Yaskawa INFORM job: DEMO_ROOF_SIDE_0625_3PAINT_51.JBI

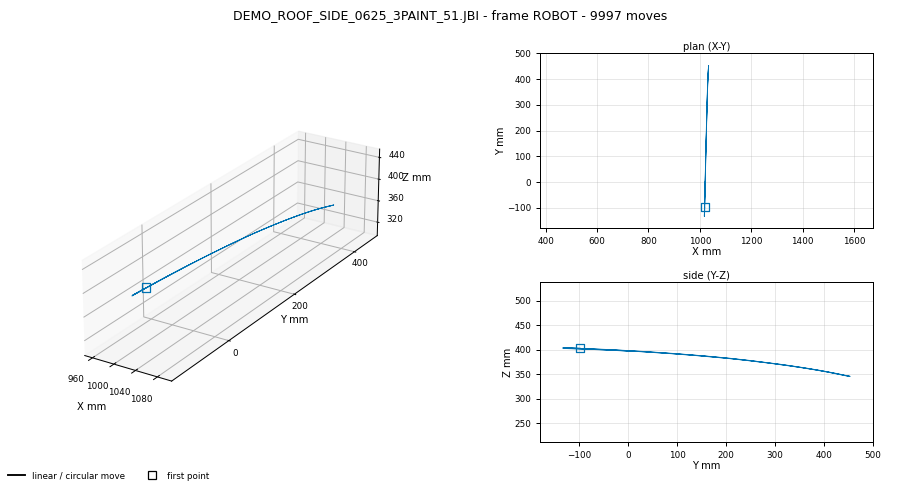
[picture p0: tool path of DEMO_ROOF_SIDE_0625_3PAINT_51.JBI in frame ROBOT, 9997 of 9997 moves have a stored position in this frame; points joined in program order, loops and branches not executed]
/JOB
//NAME DEMO_ROOF_SIDE_0625_3PAINT51
//POS
///NPOS 9997,0,0,0,0,0
///TOOL 0
///USER 0
///POSTYPE ROBOT
///RECTAN
///RCONF 1,0,0,0,0,0,0,0,0,0,0,0,0,0,0,0,0,0,0,0,0,0,0,0
C00000=1018.937,-97.840,403.399,165.576,52.819,159.418
C00001=1018.932,-98.090,403.408,165.573,52.823,159.418
C00002=1018.926,-98.340,403.416,165.570,52.828,159.419
C00003=1018.920,-98.590,403.426,165.567,52.833,159.419
C00004=1018.915,-98.839,403.434,165.564,52.838,159.419
C00005=1018.910,-99.089,403.443,165.561,52.842,159.419
C00006=1018.905,-99.339,403.452,165.558,52.848,159.420
C00007=1018.900,-99.589,403.460,165.555,52.852,159.420
C00008=1018.894,-99.839,403.469,165.552,52.857,159.420
C00009=1018.888,-100.088,403.478,165.549,52.862,159.420
C00010=1018.883,-100.338,403.487,165.546,52.867,159.420
C00011=1018.878,-100.588,403.495,165.542,52.871,159.421
C00012=1018.873,-100.837,403.504,165.540,52.876,159.421
C00013=1018.867,-101.087,403.512,165.537,52.881,159.421
C00014=1018.861,-101.371,403.523,165.534,52.887,159.421
C00015=1018.856,-101.655,403.533,165.531,52.892,159.422
C00016=1018.850,-101.939,403.543,165.526,52.897,159.422
C00017=1018.844,-102.223,403.552,165.523,52.902,159.422
C00018=1018.838,-102.472,403.561,165.520,52.908,159.422
C00019=1018.833,-102.722,403.570,165.517,52.912,159.423
C00020=1018.827,-102.972,403.579,165.514,52.917,159.423
C00021=1018.822,-103.222,403.587,165.510,52.921,159.423
C00022=1018.817,-103.472,403.596,165.508,52.927,159.423
C00023=1018.811,-103.721,403.604,165.505,52.931,159.423
C00024=1018.806,-103.971,403.613,165.501,52.936,159.424
C00025=1018.801,-104.221,403.621,165.499,52.940,159.424
C00026=1018.796,-104.471,403.630,165.496,52.946,159.424
C00027=1018.791,-104.720,403.639,165.492,52.950,159.424
C00028=1018.786,-104.970,403.647,165.490,52.955,159.425
C00029=1018.781,-105.220,403.656,165.486,52.959,159.425
C00030=1018.775,-105.470,403.664,165.483,52.965,159.425
C00031=1018.770,-105.720,403.673,165.481,52.969,159.425
C00032=1018.764,-105.970,403.681,165.477,52.974,159.425
C00033=1018.759,-106.219,403.690,165.475,52.978,159.426
C00034=1018.754,-106.469,403.698,165.472,52.984,159.426
C00035=1018.748,-106.719,403.707,165.468,52.988,159.426
C00036=1018.743,-106.969,403.715,165.466,52.993,159.426
C00037=1018.738,-107.219,403.723,165.462,52.997,159.426
C00038=1018.733,-107.469,403.732,165.459,53.003,159.427
C00039=1018.728,-107.718,403.740,165.457,53.007,159.427
C00040=1018.722,-107.968,403.749,165.453,53.012,159.427
///RCONF 1,0,0,0,1,0,0,0,0,0,0,0,0,0,0,0,0,0,0,0,0,0,0,0
C00041=1018.717,-108.218,403.757,165.450,53.017,159.427
C00042=1018.712,-108.468,403.766,165.448,53.022,159.428
C00043=1018.707,-108.718,403.773,165.444,53.026,159.428
C00044=1018.702,-108.968,403.782,165.441,53.032,159.428
C00045=1018.696,-109.217,403.790,165.439,53.036,159.428
C00046=1018.691,-109.467,403.799,165.435,53.041,159.429
C00047=1018.686,-109.717,403.807,165.432,53.045,159.429
C00048=1018.680,-109.967,403.814,165.429,53.051,159.429
C00049=1018.675,-110.216,403.823,165.426,53.055,159.429
C00050=1018.670,-110.466,403.831,165.423,53.060,159.429
C00051=1018.664,-110.716,403.840,165.420,53.065,159.430
C00052=1018.660,-110.966,403.847,165.417,53.070,159.430
C00053=1018.655,-111.215,403.856,165.414,53.074,159.430
C00054=1018.650,-111.465,403.864,165.411,53.080,159.430
C00055=1018.645,-111.715,403.872,165.408,53.084,159.431
C00056=1018.639,-111.965,403.880,165.405,53.089,159.431
C00057=1018.634,-112.215,403.889,165.401,53.094,159.431
C00058=1018.628,-112.464,403.897,165.399,53.099,159.431
C00059=1018.623,-112.714,403.905,165.396,53.103,159.431
C00060=1018.618,-112.964,403.913,165.392,53.108,159.432
C00061=1018.613,-113.214,403.922,165.390,53.112,159.432
C00062=1018.608,-113.464,403.929,165.387,53.118,159.432
C00063=1018.603,-113.713,403.938,165.384,53.122,159.432
C00064=1018.598,-113.964,403.945,165.381,53.127,159.432
C00065=1018.593,-114.213,403.954,165.377,53.132,159.433
C00066=1018.587,-114.463,403.962,165.375,53.137,159.433
C00067=1018.582,-114.713,403.969,165.372,53.141,159.433
C00068=1018.576,-114.963,403.978,165.368,53.146,159.433
C00069=1018.571,-115.213,403.986,165.366,53.151,159.434
C00070=1018.567,-115.462,403.994,165.363,53.156,159.434
C00071=1018.561,-115.712,404.001,165.359,53.161,159.434
C00072=1018.556,-115.962,404.009,165.357,53.166,159.434
C00073=1018.551,-116.212,404.018,165.354,53.170,159.435
C00074=1018.546,-116.462,404.026,165.350,53.175,159.435
C00075=1018.540,-116.711,404.033,165.347,53.180,159.435
C00076=1018.535,-116.961,404.041,165.345,53.185,159.435
C00077=1018.530,-117.211,404.049,165.341,53.190,159.435
C00078=1018.524,-117.495,404.059,165.338,53.195,159.436
C00079=1018.518,-117.779,404.067,165.335,53.201,159.436
C00080=1018.513,-118.062,404.076,165.331,53.206,159.436
C00081=1018.507,-118.346,404.085,165.328,53.211,159.436
C00082=1018.502,-118.596,404.092,165.325,53.216,159.437
C00083=1018.496,-118.846,404.101,165.322,53.221,159.437
C00084=1018.491,-119.095,404.108,165.319,53.226,159.437
C00085=1018.486,-119.345,404.116,165.316,53.231,159.437
C00086=1018.481,-119.595,404.124,165.313,53.235,159.437
C00087=1018.475,-119.845,404.131,165.310,53.240,159.438
C00088=1018.471,-120.094,404.139,165.307,53.246,159.438
C00089=1018.466,-120.345,404.147,165.304,53.250,159.438
C00090=1018.460,-120.594,404.155,165.301,53.255,159.438
C00091=1018.455,-120.844,404.163,165.297,53.259,159.438
C00092=1018.450,-121.094,404.170,165.295,53.264,159.439
C00093=1018.445,-121.344,404.179,165.292,53.269,159.439
C00094=1018.439,-121.594,404.186,165.288,53.274,159.439
C00095=1018.435,-121.843,404.193,165.286,53.278,159.439
C00096=1018.430,-122.094,404.201,165.283,53.284,159.440
C00097=1018.424,-122.343,404.209,165.279,53.288,159.440
C00098=1018.420,-122.593,404.216,165.277,53.293,159.440
C00099=1018.415,-122.843,404.224,165.274,53.298,159.440
C00100=1018.409,-123.093,404.232,165.270,53.303,159.440
C00101=1018.404,-123.342,404.239,165.268,53.307,159.441
C00102=1018.399,-123.593,404.247,165.264,53.312,159.441
C00103=1018.394,-123.843,404.254,165.261,53.318,159.441
C00104=1018.389,-124.092,404.262,165.259,53.322,159.441
C00105=1018.383,-124.342,404.269,165.255,53.327,159.441
C00106=1018.378,-124.592,404.277,165.253,53.331,159.442
C00107=1018.374,-124.842,404.285,165.250,53.337,159.442
C00108=1018.368,-125.092,404.292,165.246,53.341,159.442
C00109=1018.363,-125.342,404.300,165.244,53.346,159.442
C00110=1018.358,-125.591,404.307,165.241,53.351,159.443
C00111=1018.353,-125.841,404.315,165.238,53.356,159.443
C00112=1018.348,-126.090,404.322,165.235,53.360,159.443
C00113=1018.343,-126.341,404.329,165.232,53.366,159.443
C00114=1018.337,-126.591,404.337,165.229,53.370,159.443
C00115=1018.333,-126.840,404.344,165.225,53.375,159.443
C00116=1018.327,-127.090,404.351,165.223,53.380,159.444
C00117=1018.323,-127.340,404.359,165.220,53.385,159.444
C00118=1018.317,-127.590,404.366,165.217,53.389,159.444
C00119=1018.313,-127.839,404.374,165.214,53.394,159.444
C00120=1018.307,-128.089,404.381,165.211,53.400,159.445
C00121=1018.302,-128.339,404.389,165.208,53.403,159.445
C00122=1018.299,-128.588,404.397,165.205,53.408,159.445
C00123=1018.295,-128.837,404.406,165.202,53.410,159.445
C00124=1018.291,-129.088,404.416,165.200,53.413,159.445
C00125=1018.288,-129.337,404.426,165.196,53.416,159.444
C00126=1018.285,-129.586,404.437,165.195,53.417,159.444
C00127=1018.283,-129.836,404.448,165.192,53.418,159.444
C00128=1018.282,-130.086,404.460,165.190,53.419,159.444
C00129=1018.280,-130.336,404.473,165.187,53.419,159.443
C00130=1018.279,-130.586,404.486,165.184,53.419,159.443
C00131=1018.279,-130.836,404.500,165.182,53.418,159.442
C00132=1018.278,-131.085,404.514,165.180,53.416,159.441
C00133=1018.279,-131.334,404.529,165.178,53.414,159.440
C00134=1018.280,-131.584,404.545,165.176,53.412,159.440
C00135=1018.281,-131.834,404.560,165.174,53.408,159.438
C00136=1018.283,-132.083,404.577,165.172,53.406,159.438
C00137=1018.285,-132.333,404.594,165.170,53.401,159.436
C00138=1018.288,-132.583,404.612,165.168,53.396,159.435
C00139=1018.290,-132.833,404.631,165.167,53.391,159.434
C00140=1018.294,-133.082,404.650,165.165,53.385,159.432
C00141=1018.298,-133.332,404.669,165.164,53.379,159.431
C00142=1018.032,-133.358,404.292,165.121,53.715,159.480
C00143=1018.028,-133.109,404.273,165.123,53.722,159.482
C00144=1018.026,-132.859,404.255,165.125,53.727,159.483
C00145=1018.022,-132.610,404.236,165.127,53.732,159.485
C00146=1018.020,-132.360,404.218,165.128,53.737,159.486
C00147=1018.018,-132.110,404.201,165.130,53.742,159.487
C00148=1018.017,-131.860,404.184,165.132,53.746,159.488
C00149=1018.015,-131.610,404.168,165.134,53.748,159.489
C00150=1018.014,-131.361,404.152,165.135,53.751,159.490
C00151=1018.013,-131.111,404.137,165.138,53.753,159.490
C00152=1018.014,-130.861,404.123,165.140,53.754,159.491
C00153=1018.014,-130.611,404.109,165.142,53.755,159.492
C00154=1018.015,-130.362,404.096,165.145,53.755,159.492
C00155=1018.016,-130.112,404.084,165.147,53.755,159.493
C00156=1018.018,-129.862,404.072,165.150,53.755,159.493
C00157=1018.020,-129.613,404.060,165.153,53.754,159.494
C00158=1018.023,-129.363,404.050,165.154,53.752,159.494
C00159=1018.026,-129.113,404.039,165.158,53.749,159.494
C00160=1018.029,-128.864,404.030,165.160,53.747,159.494
C00161=1018.033,-128.614,404.021,165.163,53.743,159.494
C00162=1018.037,-128.365,404.012,165.166,53.739,159.494
C00163=1018.042,-128.115,404.004,165.168,53.735,159.494
C00164=1018.046,-127.866,403.996,165.172,53.730,159.494
C00165=1018.052,-127.616,403.989,165.175,53.725,159.494
C00166=1018.057,-127.366,403.982,165.178,53.720,159.493
C00167=1018.061,-127.117,403.975,165.180,53.716,159.493
C00168=1018.067,-126.867,403.968,165.183,53.710,159.493
C00169=1018.072,-126.616,403.960,165.187,53.705,159.493
C00170=1018.077,-126.367,403.953,165.190,53.700,159.493
C00171=1018.082,-126.117,403.945,165.192,53.695,159.492
C00172=1018.087,-125.867,403.939,165.196,53.691,159.492
C00173=1018.092,-125.617,403.931,165.199,53.685,159.492
C00174=1018.098,-125.368,403.923,165.202,53.680,159.492
C00175=1018.103,-125.118,403.915,165.204,53.675,159.491
C00176=1018.108,-124.868,403.908,165.208,53.670,159.491
C00177=1018.113,-124.618,403.901,165.211,53.666,159.491
C00178=1018.118,-124.368,403.893,165.214,53.660,159.491
C00179=1018.123,-124.119,403.886,165.216,53.656,159.490
C00180=1018.128,-123.868,403.879,165.220,53.651,159.490
C00181=1018.133,-123.619,403.870,165.223,53.645,159.490
C00182=1018.138,-123.369,403.863,165.225,53.641,159.490
C00183=1018.143,-123.119,403.856,165.229,53.636,159.490
C00184=1018.148,-122.869,403.848,165.232,53.631,159.489
C00185=1018.153,-122.620,403.840,165.235,53.626,159.489
C00186=1018.158,-122.370,403.832,165.237,53.621,159.489
C00187=1018.163,-122.119,403.825,165.241,53.616,159.489
C00188=1018.168,-121.870,403.818,165.244,53.611,159.489
C00189=1018.174,-121.620,403.809,165.246,53.606,159.488
C00190=1018.179,-121.370,403.802,165.249,53.602,159.488
C00191=1018.184,-121.121,403.795,165.253,53.597,159.488
C00192=1018.189,-120.870,403.787,165.256,53.591,159.488
C00193=1018.194,-120.621,403.779,165.258,53.587,159.487
C00194=1018.199,-120.371,403.772,165.261,53.581,159.487
C00195=1018.207,-119.987,403.759,165.266,53.574,159.487
C00196=1018.215,-119.603,403.748,165.271,53.566,159.487
C00197=1018.223,-119.219,403.735,165.275,53.559,159.486
C00198=1018.231,-118.835,403.724,165.280,53.551,159.486
C00199=1018.239,-118.435,403.711,165.285,53.543,159.485
C00200=1018.247,-118.037,403.699,165.289,53.535,159.485
C00201=1018.255,-117.637,403.686,165.294,53.527,159.485
C00202=1018.264,-117.238,403.674,165.299,53.520,159.484
C00203=1018.268,-116.988,403.666,165.302,53.515,159.484
C00204=1018.273,-116.738,403.658,165.306,53.510,159.484
C00205=1018.279,-116.488,403.650,165.309,53.505,159.484
C00206=1018.284,-116.238,403.643,165.311,53.500,159.483
C00207=1018.289,-115.988,403.634,165.314,53.495,159.483
C00208=1018.294,-115.739,403.627,165.317,53.490,159.483
C00209=1018.300,-115.489,403.619,165.321,53.485,159.483
C00210=1018.305,-115.239,403.611,165.323,53.480,159.482
C00211=1018.310,-114.989,403.603,165.326,53.475,159.482
C00212=1018.315,-114.739,403.595,165.329,53.470,159.482
C00213=1018.320,-114.490,403.587,165.333,53.465,159.482
C00214=1018.325,-114.241,403.579,165.335,53.461,159.482
C00215=1018.330,-113.990,403.571,165.338,53.455,159.481
C00216=1018.336,-113.740,403.563,165.342,53.451,159.481
C00217=1018.341,-113.490,403.555,165.345,53.445,159.481
C00218=1018.346,-113.240,403.546,165.347,53.441,159.481
C00219=1018.351,-112.991,403.538,165.351,53.436,159.480
C00220=1018.355,-112.741,403.530,165.354,53.431,159.480
C00221=1018.361,-112.491,403.522,165.356,53.426,159.480
C00222=1018.367,-112.242,403.514,165.359,53.422,159.480
C00223=1018.372,-111.992,403.506,165.363,53.416,159.479
C00224=1018.377,-111.742,403.498,165.366,53.411,159.479
C00225=1018.382,-111.492,403.489,165.368,53.407,159.479
C00226=1018.387,-111.242,403.482,165.371,53.401,159.479
C00227=1018.392,-110.992,403.473,165.375,53.397,159.479
C00228=1018.398,-110.742,403.465,165.378,53.391,159.478
C00229=1018.402,-110.493,403.457,165.380,53.387,159.478
C00230=1018.407,-110.243,403.449,165.384,53.382,159.478
C00231=1018.413,-109.994,403.441,165.387,53.377,159.478
C00232=1018.418,-109.743,403.433,165.390,53.372,159.477
C00233=1018.424,-109.494,403.425,165.392,53.367,159.477
C00234=1018.429,-109.244,403.416,165.396,53.362,159.477
C00235=1018.434,-108.994,403.408,165.399,53.357,159.477
C00236=1018.439,-108.744,403.400,165.402,53.352,159.476
C00237=1018.444,-108.494,403.391,165.405,53.348,159.476
C00238=1018.450,-108.244,403.383,165.408,53.342,159.476
C00239=1018.455,-107.995,403.374,165.411,53.337,159.476
C00240=1018.460,-107.745,403.366,165.414,53.332,159.475
C00241=1018.465,-107.495,403.358,165.417,53.328,159.475
C00242=1018.470,-107.245,403.350,165.420,53.323,159.475
C00243=1018.476,-106.995,403.341,165.423,53.317,159.475
C00244=1018.481,-106.745,403.333,165.427,53.313,159.475
C00245=1018.486,-106.496,403.324,165.429,53.308,159.474
///RCONF 1,0,0,0,0,0,0,0,0,0,0,0,0,0,0,0,0,0,0,0,0,0,0,0
C00246=1018.491,-106.246,403.316,165.432,53.303,159.474
C00247=1018.497,-105.996,403.307,165.435,53.298,159.474
C00248=1018.502,-105.747,403.299,165.439,53.293,159.474
C00249=1018.507,-105.497,403.290,165.441,53.288,159.473
C00250=1018.512,-105.247,403.282,165.444,53.284,159.473
C00251=1018.517,-104.997,403.274,165.447,53.278,159.473
C00252=1018.523,-104.747,403.266,165.450,53.274,159.473
C00253=1018.528,-104.497,403.257,165.453,53.269,159.473
C00254=1018.533,-104.248,403.249,165.456,53.264,159.472
C00255=1018.538,-103.998,403.240,165.460,53.259,159.472
C00256=1018.543,-103.748,403.231,165.462,53.255,159.472
C00257=1018.548,-103.498,403.222,165.465,53.249,159.471
C00258=1018.554,-103.249,403.214,165.469,53.244,159.471
C00259=1018.559,-102.998,403.205,165.472,53.239,159.471
C00260=1018.565,-102.748,403.197,165.474,53.235,159.471
C00261=1018.570,-102.499,403.188,165.478,53.230,159.471
C00262=1018.575,-102.249,403.180,165.481,53.224,159.470
C00263=1018.581,-101.965,403.170,165.484,53.219,159.470
C00264=1018.587,-101.682,403.160,165.488,53.213,159.470
C00265=1018.593,-101.398,403.150,165.491,53.208,159.469
C00266=1018.599,-101.115,403.140,165.494,53.202,159.469
C00267=1018.604,-100.865,403.132,165.497,53.198,159.469
C00268=1018.610,-100.615,403.123,165.500,53.192,159.469
C00269=1018.615,-100.365,403.114,165.504,53.187,159.469
C00270=1018.620,-100.115,403.105,165.506,53.183,159.468
C00271=1018.625,-99.865,403.097,165.509,53.178,159.468
C00272=1018.631,-99.616,403.088,165.513,53.173,159.468
C00273=1018.636,-99.366,403.079,165.516,53.167,159.468
C00274=1018.641,-99.117,403.071,165.518,53.163,159.467
C00275=1018.647,-98.866,403.062,165.521,53.158,159.467
C00276=1018.652,-98.617,403.053,165.525,53.153,159.467
C00277=1018.657,-98.367,403.044,165.528,53.148,159.467
C00278=1018.663,-98.117,403.035,165.530,53.143,159.466
C00279=1018.668,-97.868,403.026,165.534,53.138,159.466
C00280=1018.674,-97.617,403.018,165.537,53.133,159.466
C00281=1018.678,-97.367,403.009,165.539,53.129,159.465
C00282=1018.684,-97.118,402.999,165.543,53.124,159.465
C00283=1018.689,-96.868,402.991,165.546,53.119,159.465
C00284=1018.694,-96.618,402.982,165.548,53.114,159.465
C00285=1018.700,-96.369,402.972,165.552,53.109,159.465
C00286=1018.704,-96.119,402.963,165.555,53.105,159.465
C00287=1018.710,-95.869,402.955,165.558,53.100,159.464
C00288=1018.714,-95.620,402.945,165.561,53.095,159.464
C00289=1018.720,-95.369,402.936,165.564,53.090,159.464
C00290=1018.725,-95.119,402.928,165.567,53.086,159.464
C00291=1018.730,-94.870,402.918,165.570,53.081,159.463
C00292=1018.736,-94.620,402.909,165.573,53.076,159.463
C00293=1018.741,-94.370,402.899,165.576,53.072,159.463
C00294=1018.746,-94.120,402.891,165.579,53.067,159.463
C00295=1018.752,-93.871,402.881,165.582,53.061,159.462
C00296=1018.756,-93.621,402.872,165.586,53.057,159.462
C00297=1018.762,-93.371,402.863,165.588,53.052,159.462
C00298=1018.767,-93.121,402.854,165.591,53.047,159.462
C00299=1018.772,-92.872,402.845,165.595,53.042,159.461
C00300=1018.779,-92.622,402.836,165.597,53.038,159.461
C00301=1018.783,-92.372,402.827,165.600,53.032,159.461
C00302=1018.789,-92.123,402.817,165.604,53.028,159.461
C00303=1018.794,-91.872,402.808,165.606,53.023,159.460
C00304=1018.799,-91.623,402.799,165.609,53.018,159.460
C00305=1018.804,-91.373,402.790,165.613,53.013,159.460
C00306=1018.810,-91.123,402.780,165.615,53.009,159.460
C00307=1018.815,-90.873,402.772,165.618,53.004,159.459
C00308=1018.820,-90.624,402.762,165.622,52.999,159.459
C00309=1018.826,-90.374,402.753,165.625,52.993,159.459
C00310=1018.831,-90.124,402.743,165.627,52.989,159.459
C00311=1018.836,-89.875,402.735,165.631,52.984,159.459
C00312=1018.841,-89.624,402.724,165.634,52.979,159.458
C00313=1018.847,-89.375,402.715,165.636,52.975,159.458
C00314=1018.852,-89.126,402.707,165.640,52.970,159.458
C00315=1018.858,-88.876,402.697,165.643,52.965,159.457
C00316=1018.863,-88.626,402.688,165.646,52.960,159.457
C00317=1018.868,-88.376,402.678,165.648,52.955,159.457
C00318=1018.874,-88.127,402.669,165.652,52.950,159.457
C00319=1018.879,-87.876,402.659,165.655,52.945,159.457
C00320=1018.885,-87.627,402.650,165.658,52.940,159.456
C00321=1018.890,-87.377,402.642,165.661,52.936,159.456
C00322=1018.895,-87.127,402.631,165.664,52.930,159.456
C00323=1018.901,-86.878,402.622,165.667,52.926,159.456
C00324=1018.906,-86.627,402.613,165.669,52.921,159.455
C00325=1018.912,-86.378,402.604,165.673,52.916,159.455
C00326=1018.917,-86.128,402.593,165.676,52.911,159.455
C00327=1018.924,-85.846,402.584,165.679,52.905,159.454
C00328=1018.930,-85.564,402.573,165.683,52.899,159.454
C00329=1018.935,-85.284,402.562,165.686,52.894,159.454
C00330=1018.942,-85.002,402.552,165.689,52.889,159.453
C00331=1018.947,-84.752,402.542,165.692,52.884,159.453
C00332=1018.952,-84.503,402.533,165.696,52.878,159.453
C00333=1018.958,-84.252,402.523,165.699,52.874,159.453
C00334=1018.963,-84.003,402.514,165.701,52.869,159.452
C00335=1018.969,-83.753,402.504,165.705,52.864,159.452
C00336=1018.974,-83.504,402.495,165.708,52.859,159.452
C00337=1018.979,-83.253,402.485,165.711,52.854,159.452
C00338=1018.986,-83.004,402.476,165.714,52.850,159.451
C00339=1018.991,-82.755,402.466,165.717,52.844,159.451
C00340=1018.996,-82.504,402.457,165.720,52.840,159.451
C00341=1019.002,-82.255,402.448,165.723,52.834,159.451
C00342=1019.007,-82.005,402.438,165.725,52.829,159.450
C00343=1019.013,-81.755,402.428,165.729,52.824,159.450
C00344=1019.018,-81.505,402.418,165.732,52.819,159.450
C00345=1019.024,-81.256,402.410,165.735,52.814,159.449
C00346=1019.029,-81.006,402.400,165.737,52.809,159.449
C00347=1019.035,-80.756,402.390,165.741,52.805,159.449
C00348=1019.040,-80.506,402.380,165.744,52.799,159.448
C00349=1019.046,-80.257,402.371,165.747,52.795,159.448
C00350=1019.051,-80.007,402.361,165.749,52.790,159.448
C00351=1019.056,-79.757,402.351,165.753,52.785,159.448
C00352=1019.063,-79.507,402.341,165.756,52.780,159.448
C00353=1019.067,-79.258,402.331,165.758,52.775,159.447
C00354=1019.073,-79.008,402.321,165.762,52.771,159.447
C00355=1019.078,-78.758,402.311,165.765,52.766,159.447
C00356=1019.084,-78.508,402.302,165.768,52.760,159.446
C00357=1019.089,-78.258,402.292,165.771,52.756,159.446
C00358=1019.094,-78.009,402.282,165.774,52.751,159.446
C00359=1019.100,-77.759,402.272,165.777,52.746,159.446
C00360=1019.105,-77.510,402.262,165.780,52.742,159.445
C00361=1019.111,-77.260,402.252,165.783,52.736,159.445
C00362=1019.116,-77.010,402.242,165.787,52.732,159.445
C00363=1019.122,-76.760,402.233,165.789,52.727,159.445
C00364=1019.127,-76.510,402.223,165.792,52.722,159.444
C00365=1019.132,-76.260,402.213,165.796,52.717,159.444
C00366=1019.137,-76.011,402.203,165.798,52.712,159.444
C00367=1019.143,-75.761,402.193,165.801,52.708,159.444
C00368=1019.149,-75.512,402.182,165.804,52.702,159.443
C00369=1019.154,-75.262,402.173,165.807,52.698,159.443
C00370=1019.159,-75.012,402.162,165.810,52.693,159.443
C00371=1019.166,-74.762,402.153,165.813,52.688,159.442
C00372=1019.171,-74.512,402.143,165.817,52.683,159.442
C00373=1019.176,-74.263,402.133,165.819,52.678,159.442
C00374=1019.182,-74.013,402.122,165.822,52.674,159.442
C00375=1019.187,-73.763,402.112,165.825,52.669,159.441
C00376=1019.192,-73.514,402.102,165.828,52.665,159.441
C00377=1019.198,-73.264,402.091,165.831,52.659,159.441
C00378=1019.203,-73.014,402.081,165.834,52.655,159.441
C00379=1019.209,-72.764,402.071,165.837,52.650,159.440
C00380=1019.214,-72.515,402.060,165.840,52.646,159.440
C00381=1019.219,-72.265,402.050,165.843,52.641,159.440
C00382=1019.225,-72.015,402.040,165.845,52.636,159.440
C00383=1019.230,-71.766,402.029,165.849,52.632,159.439
C00384=1019.234,-71.516,402.019,165.852,52.627,159.439
C00385=1019.240,-71.266,402.009,165.854,52.622,159.439
C00386=1019.246,-71.016,401.998,165.858,52.617,159.439
C00387=1019.251,-70.766,401.988,165.860,52.613,159.438
C00388=1019.256,-70.517,401.978,165.864,52.608,159.438
C00389=1019.262,-70.267,401.967,165.867,52.603,159.438
C00390=1019.267,-70.017,401.957,165.869,52.599,159.438
C00391=1019.273,-69.737,401.945,165.872,52.593,159.437
C00392=1019.280,-69.458,401.933,165.877,52.588,159.437
C00393=1019.286,-69.179,401.921,165.880,52.582,159.437
C00394=1019.291,-68.898,401.910,165.883,52.578,159.436
C00395=1019.297,-68.650,401.899,165.886,52.572,159.436
C00396=1019.302,-68.399,401.889,165.889,52.568,159.436
C00397=1019.308,-68.150,401.878,165.892,52.563,159.436
C00398=1019.313,-67.900,401.868,165.894,52.558,159.435
C00399=1019.319,-67.650,401.857,165.898,52.554,159.435
C00400=1019.324,-67.400,401.847,165.901,52.549,159.435
C00401=1019.329,-67.151,401.837,165.903,52.544,159.434
C00402=1019.335,-66.901,401.826,165.907,52.539,159.434
C00403=1019.341,-66.652,401.816,165.910,52.535,159.434
C00404=1019.346,-66.402,401.805,165.912,52.530,159.434
C00405=1019.351,-66.152,401.794,165.916,52.525,159.433
C00406=1019.356,-65.902,401.784,165.918,52.520,159.433
C00407=1019.362,-65.652,401.773,165.922,52.516,159.433
C00408=1019.368,-65.402,401.763,165.925,52.511,159.433
C00409=1019.373,-65.153,401.752,165.927,52.506,159.432
C00410=1019.379,-64.904,401.741,165.931,52.501,159.432
C00411=1019.384,-64.654,401.731,165.934,52.496,159.432
C00412=1019.390,-64.404,401.720,165.936,52.492,159.431
C00413=1019.395,-64.154,401.710,165.939,52.486,159.431
C00414=1019.401,-63.905,401.699,165.943,52.482,159.431
C00415=1019.407,-63.655,401.688,165.945,52.477,159.431
C00416=1019.412,-63.405,401.678,165.948,52.472,159.430
C00417=1019.418,-63.156,401.667,165.952,52.467,159.430
C00418=1019.423,-62.906,401.657,165.954,52.462,159.430
C00419=1019.428,-62.656,401.646,165.957,52.458,159.429
C00420=1019.434,-62.406,401.635,165.961,52.452,159.429
C00421=1019.439,-62.156,401.625,165.963,52.448,159.429
C00422=1019.445,-61.907,401.614,165.966,52.443,159.428
C00423=1019.451,-61.657,401.603,165.970,52.438,159.428
C00424=1019.456,-61.407,401.593,165.972,52.433,159.428
C00425=1019.462,-61.158,401.582,165.975,52.428,159.428
C00426=1019.468,-60.908,401.571,165.978,52.423,159.427
C00427=1019.473,-60.658,401.561,165.981,52.419,159.427
C00428=1019.479,-60.409,401.550,165.984,52.413,159.427
C00429=1019.485,-60.159,401.539,165.987,52.409,159.426
C00430=1019.490,-59.909,401.528,165.989,52.404,159.426
C00431=1019.495,-59.659,401.518,165.993,52.399,159.426
C00432=1019.501,-59.410,401.507,165.996,52.394,159.425
C00433=1019.507,-59.160,401.496,165.999,52.390,159.425
C00434=1019.512,-58.911,401.485,166.002,52.384,159.425
C00435=1019.518,-58.661,401.475,166.005,52.379,159.424
C00436=1019.523,-58.411,401.464,166.008,52.374,159.424
C00437=1019.529,-58.162,401.453,166.010,52.369,159.424
C00438=1019.535,-57.912,401.442,166.014,52.365,159.424
C00439=1019.540,-57.662,401.432,166.017,52.359,159.423
C00440=1019.545,-57.412,401.420,166.019,52.355,159.423
C00441=1019.551,-57.163,401.410,166.023,52.350,159.423
C00442=1019.557,-56.913,401.399,166.026,52.344,159.422
C00443=1019.563,-56.664,401.388,166.029,52.340,159.422
C00444=1019.568,-56.414,401.378,166.031,52.335,159.422
C00445=1019.574,-56.164,401.367,166.035,52.330,159.421
C00446=1019.580,-55.914,401.356,166.038,52.325,159.421
C00447=1019.586,-55.664,401.345,166.040,52.320,159.421
C00448=1019.592,-55.415,401.334,166.043,52.315,159.420
C00449=1019.597,-55.165,401.322,166.047,52.310,159.420
C00450=1019.602,-54.916,401.311,166.050,52.305,159.420
C00451=1019.608,-54.666,401.301,166.052,52.300,159.419
C00452=1019.614,-54.416,401.290,166.055,52.295,159.419
C00453=1019.619,-54.167,401.280,166.058,52.290,159.419
C00454=1019.626,-53.916,401.268,166.061,52.285,159.418
C00455=1019.631,-53.638,401.256,166.065,52.279,159.418
C00456=1019.638,-53.359,401.244,166.068,52.274,159.418
C00457=1019.645,-53.082,401.232,166.071,52.268,159.417
C00458=1019.651,-52.803,401.219,166.075,52.263,159.417
C00459=1019.657,-52.553,401.208,166.077,52.258,159.416
C00460=1019.663,-52.304,401.197,166.080,52.252,159.416
C00461=1019.668,-52.054,401.187,166.084,52.248,159.416
C00462=1019.674,-51.805,401.176,166.087,52.242,159.416
C00463=1019.680,-51.554,401.164,166.089,52.237,159.415
C00464=1019.685,-51.305,401.153,166.092,52.232,159.415
C00465=1019.691,-51.055,401.142,166.096,52.228,159.415
C00466=1019.697,-50.806,401.131,166.098,52.223,159.414
C00467=1019.702,-50.556,401.120,166.101,52.218,159.414
C00468=1019.708,-50.306,401.109,166.104,52.213,159.414
C00469=1019.713,-50.056,401.097,166.107,52.208,159.413
C00470=1019.719,-49.807,401.085,166.110,52.203,159.413
C00471=1019.724,-49.557,401.074,166.112,52.199,159.413
C00472=1019.730,-49.308,401.063,166.115,52.193,159.412
C00473=1019.736,-49.057,401.051,166.119,52.189,159.412
C00474=1019.741,-48.808,401.040,166.121,52.184,159.412
C00475=1019.747,-48.558,401.028,166.125,52.179,159.411
C00476=1019.752,-48.309,401.017,166.127,52.174,159.411
C00477=1019.758,-48.058,401.006,166.130,52.170,159.411
C00478=1019.764,-47.809,400.995,166.133,52.164,159.410
C00479=1019.769,-47.560,400.982,166.136,52.160,159.410
C00480=1019.775,-47.310,400.972,166.139,52.155,159.410
C00481=1019.780,-47.060,400.960,166.142,52.150,159.410
C00482=1019.786,-46.811,400.948,166.145,52.145,159.409
C00483=1019.791,-46.561,400.937,166.148,52.141,159.409
C00484=1019.797,-46.311,400.925,166.150,52.136,159.408
C00485=1019.803,-46.061,400.914,166.154,52.131,159.408
C00486=1019.808,-45.812,400.902,166.157,52.126,159.408
C00487=1019.814,-45.562,400.891,166.159,52.121,159.407
C00488=1019.819,-45.312,400.879,166.162,52.116,159.407
C00489=1019.825,-45.063,400.867,166.166,52.111,159.407
C00490=1019.830,-44.813,400.856,166.168,52.107,159.406
C00491=1019.837,-44.563,400.845,166.171,52.101,159.406
C00492=1019.842,-44.314,400.833,166.174,52.097,159.406
C00493=1019.848,-44.064,400.822,166.177,52.092,159.405
C00494=1019.854,-43.815,400.809,166.180,52.086,159.405
C00495=1019.859,-43.565,400.798,166.182,52.082,159.405
C00496=1019.864,-43.315,400.787,166.186,52.077,159.404
C00497=1019.870,-43.065,400.774,166.189,52.072,159.404
C00498=1019.876,-42.816,400.763,166.191,52.067,159.404
C00499=1019.881,-42.566,400.752,166.194,52.062,159.403
C00500=1019.888,-42.317,400.740,166.197,52.057,159.403
C00501=1019.893,-42.067,400.728,166.200,52.053,159.403
C00502=1019.899,-41.817,400.716,166.203,52.047,159.402
C00503=1019.904,-41.567,400.705,166.206,52.042,159.402
C00504=1019.910,-41.318,400.693,166.209,52.038,159.402
C00505=1019.916,-41.068,400.682,166.212,52.032,159.401
C00506=1019.921,-40.819,400.669,166.215,52.027,159.401
C00507=1019.928,-40.569,400.658,166.217,52.023,159.401
C00508=1019.933,-40.319,400.646,166.221,52.018,159.400
C00509=1019.939,-40.070,400.635,166.224,52.012,159.400
C00510=1019.944,-39.819,400.623,166.226,52.008,159.400
C00511=1019.950,-39.571,400.612,166.229,52.003,159.399
C00512=1019.956,-39.320,400.600,166.232,51.997,159.399
C00513=1019.961,-39.071,400.588,166.235,51.993,159.398
C00514=1019.968,-38.821,400.576,166.238,51.988,159.398
C00515=1019.973,-38.572,400.564,166.241,51.984,159.398
C00516=1019.979,-38.322,400.552,166.244,51.978,159.397
C00517=1019.984,-38.072,400.539,166.247,51.973,159.397
C00518=1019.989,-37.823,400.528,166.249,51.969,159.397
C00519=1019.996,-37.544,400.515,166.253,51.964,159.396
C00520=1020.002,-37.266,400.501,166.256,51.958,159.396
C00521=1020.008,-36.988,400.488,166.259,51.953,159.396
C00522=1020.015,-36.710,400.475,166.263,51.947,159.395
C00523=1020.020,-36.461,400.462,166.265,51.942,159.395
C00524=1020.026,-36.211,400.450,166.268,51.937,159.395
C00525=1020.031,-35.961,400.438,166.271,51.933,159.394
C00526=1020.037,-35.711,400.426,166.274,51.928,159.394
C00527=1020.043,-35.462,400.414,166.276,51.923,159.393
C00528=1020.049,-35.212,400.402,166.280,51.918,159.393
C00529=1020.054,-34.963,400.390,166.283,51.913,159.393
C00530=1020.060,-34.713,400.378,166.285,51.909,159.392
C00531=1020.065,-34.464,400.365,166.288,51.903,159.392
C00532=1020.071,-34.213,400.354,166.290,51.898,159.392
C00533=1020.077,-33.964,400.342,166.294,51.894,159.391
C00534=1020.083,-33.714,400.329,166.297,51.888,159.391
C00535=1020.089,-33.464,400.317,166.299,51.884,159.391
C00536=1020.094,-33.215,400.305,166.303,51.879,159.390
C00537=1020.100,-32.965,400.293,166.306,51.874,159.390
C00538=1020.105,-32.716,400.281,166.308,51.869,159.389
C00539=1020.112,-32.466,400.269,166.312,51.864,159.389
C00540=1020.117,-32.217,400.257,166.314,51.859,159.389
C00541=1020.123,-31.967,400.244,166.317,51.854,159.388
C00542=1020.128,-31.718,400.232,166.320,51.849,159.388
C00543=1020.134,-31.467,400.220,166.322,51.844,159.388
C00544=1020.140,-31.217,400.207,166.326,51.839,159.387
C00545=1020.146,-30.969,400.196,166.328,51.834,159.387
C00546=1020.152,-30.719,400.183,166.331,51.830,159.387
C00547=1020.157,-30.469,400.171,166.334,51.824,159.386
C00548=1020.163,-30.220,400.159,166.337,51.820,159.386
C00549=1020.169,-29.970,400.146,166.340,51.814,159.385
C00550=1020.174,-29.720,400.134,166.343,51.810,159.385
C00551=1020.180,-29.470,400.122,166.345,51.805,159.385
C00552=1020.186,-29.221,400.110,166.348,51.799,159.384
C00553=1020.192,-28.971,400.098,166.352,51.794,159.384
C00554=1020.198,-28.721,400.085,166.354,51.790,159.384
C00555=1020.203,-28.472,400.073,166.357,51.785,159.383
C00556=1020.209,-28.222,400.060,166.359,51.780,159.383
C00557=1020.215,-27.972,400.048,166.363,51.775,159.382
C00558=1020.220,-27.723,400.036,166.366,51.769,159.382
C00559=1020.226,-27.473,400.023,166.368,51.765,159.382
C00560=1020.232,-27.223,400.011,166.371,51.760,159.381
C00561=1020.237,-26.974,399.998,166.374,51.755,159.381
C00562=1020.243,-26.724,399.986,166.377,51.750,159.381
C00563=1020.249,-26.475,399.973,166.379,51.745,159.380
C00564=1020.255,-26.225,399.961,166.382,51.740,159.380
C00565=1020.260,-25.975,399.949,166.386,51.736,159.380
C00566=1020.266,-25.726,399.936,166.388,51.731,159.379
C00567=1020.272,-25.476,399.922,166.392,51.726,159.379
C00568=1020.277,-25.227,399.910,166.394,51.721,159.378
C00569=1020.283,-24.977,399.897,166.397,51.716,159.378
C00570=1020.289,-24.727,399.885,166.399,51.712,159.378
C00571=1020.294,-24.478,399.873,166.403,51.706,159.377
C00572=1020.300,-24.228,399.860,166.405,51.702,159.377
C00573=1020.306,-23.979,399.847,166.408,51.696,159.376
C00574=1020.311,-23.730,399.835,166.411,51.692,159.376
C00575=1020.317,-23.479,399.822,166.413,51.687,159.376
C00576=1020.322,-23.229,399.809,166.417,51.682,159.375
C00577=1020.328,-22.980,399.796,166.419,51.677,159.375
C00578=1020.334,-22.731,399.784,166.422,51.672,159.375
C00579=1020.340,-22.481,399.771,166.424,51.667,159.374
C00580=1020.346,-22.231,399.758,166.428,51.662,159.374
C00581=1020.352,-21.981,399.746,166.431,51.657,159.373
C00582=1020.356,-21.732,399.733,166.433,51.652,159.373
C00583=1020.364,-21.453,399.719,166.436,51.647,159.373
C00584=1020.370,-21.174,399.704,166.439,51.641,159.372
C00585=1020.376,-20.895,399.690,166.442,51.636,159.372
C00586=1020.383,-20.616,399.676,166.447,51.630,159.371
C00587=1020.388,-20.366,399.663,166.449,51.625,159.371
C00588=1020.394,-20.116,399.651,166.452,51.620,159.370
C00589=1020.400,-19.868,399.638,166.454,51.615,159.370
C00590=1020.406,-19.618,399.625,166.457,51.610,159.370
C00591=1020.411,-19.368,399.612,166.461,51.606,159.369
C00592=1020.417,-19.118,399.599,166.463,51.601,159.369
C00593=1020.423,-18.868,399.586,166.466,51.595,159.368
C00594=1020.429,-18.619,399.574,166.468,51.590,159.368
C00595=1020.435,-18.370,399.561,166.471,51.585,159.368
C00596=1020.441,-18.120,399.548,166.475,51.581,159.367
C00597=1020.447,-17.870,399.536,166.477,51.576,159.367
C00598=1020.452,-17.621,399.522,166.480,51.571,159.366
C00599=1020.458,-17.371,399.509,166.482,51.566,159.366
C00600=1020.463,-17.122,399.497,166.486,51.560,159.366
C00601=1020.469,-16.872,399.484,166.489,51.555,159.365
C00602=1020.475,-16.623,399.471,166.491,51.550,159.365
C00603=1020.481,-16.373,399.459,166.494,51.546,159.364
C00604=1020.487,-16.123,399.445,166.497,51.541,159.364
C00605=1020.493,-15.873,399.432,166.500,51.536,159.364
C00606=1020.499,-15.624,399.419,166.502,51.531,159.363
C00607=1020.504,-15.374,399.406,166.505,51.525,159.363
C00608=1020.510,-15.125,399.393,166.508,51.521,159.362
C00609=1020.516,-14.875,399.380,166.511,51.516,159.362
C00610=1020.521,-14.626,399.366,166.514,51.511,159.362
C00611=1020.527,-14.376,399.354,166.516,51.506,159.361
C00612=1020.532,-14.126,399.340,166.520,51.501,159.361
C00613=1020.539,-13.877,399.327,166.522,51.496,159.360
C00614=1020.544,-13.627,399.314,166.525,51.491,159.360
C00615=1020.550,-13.378,399.300,166.527,51.486,159.359
C00616=1020.556,-13.128,399.288,166.531,51.482,159.359
C00617=1020.561,-12.878,399.274,166.533,51.477,159.359
C00618=1020.567,-12.629,399.261,166.536,51.472,159.358
C00619=1020.572,-12.379,399.248,166.538,51.467,159.358
C00620=1020.578,-12.130,399.235,166.542,51.462,159.358
C00621=1020.584,-11.880,399.221,166.544,51.457,159.357
C00622=1020.590,-11.631,399.208,166.547,51.452,159.357
C00623=1020.596,-11.381,399.195,166.549,51.447,159.356
C00624=1020.601,-11.131,399.182,166.552,51.442,159.356
C00625=1020.607,-10.882,399.168,166.555,51.438,159.356
C00626=1020.613,-10.632,399.155,166.558,51.433,159.355
C00627=1020.619,-10.382,399.142,166.561,51.427,159.355
C00628=1020.624,-10.133,399.128,166.563,51.423,159.354
C00629=1020.630,-9.884,399.115,166.567,51.417,159.354
C00630=1020.636,-9.633,399.102,166.569,51.412,159.353
C00631=1020.642,-9.384,399.089,166.572,51.408,159.353
C00632=1020.648,-9.135,399.075,166.574,51.403,159.353
C00633=1020.653,-8.885,399.062,166.578,51.398,159.352
C00634=1020.659,-8.635,399.049,166.580,51.393,159.352
C00635=1020.665,-8.386,399.035,166.583,51.388,159.351
C00636=1020.671,-8.137,399.022,166.585,51.383,159.351
C00637=1020.676,-7.886,399.009,166.588,51.378,159.350
C00638=1020.683,-7.637,398.995,166.591,51.372,159.350
C00639=1020.688,-7.387,398.981,166.594,51.368,159.350
C00640=1020.694,-7.138,398.968,166.597,51.363,159.349
C00641=1020.700,-6.888,398.956,166.599,51.358,159.349
C00642=1020.706,-6.639,398.942,166.602,51.353,159.348
C00643=1020.712,-6.390,398.928,166.605,51.348,159.348
C00644=1020.717,-6.140,398.915,166.608,51.343,159.347
C00645=1020.723,-5.890,398.902,166.611,51.338,159.347
C00646=1020.729,-5.640,398.888,166.613,51.333,159.347
C00647=1020.736,-5.360,398.873,166.616,51.327,159.346
C00648=1020.743,-5.079,398.858,166.619,51.322,159.346
C00649=1020.749,-4.798,398.843,166.623,51.315,159.345
C00650=1020.756,-4.517,398.827,166.626,51.310,159.345
C00651=1020.762,-4.268,398.814,166.628,51.305,159.344
C00652=1020.767,-4.018,398.800,166.632,51.300,159.344
C00653=1020.773,-3.769,398.786,166.634,51.295,159.343
C00654=1020.778,-3.519,398.772,166.637,51.291,159.343
C00655=1020.784,-3.270,398.759,166.639,51.286,159.343
C00656=1020.790,-3.020,398.745,166.643,51.281,159.342
C00657=1020.795,-2.771,398.731,166.645,51.276,159.342
C00658=1020.801,-2.521,398.718,166.647,51.271,159.341
C00659=1020.806,-2.272,398.704,166.651,51.266,159.341
C00660=1020.812,-2.022,398.690,166.653,51.261,159.340
C00661=1020.819,-1.772,398.676,166.656,51.256,159.340
C00662=1020.824,-1.522,398.662,166.658,51.251,159.339
C00663=1020.830,-1.273,398.648,166.662,51.247,159.339
C00664=1020.835,-1.023,398.635,166.664,51.242,159.339
C00665=1020.841,-0.774,398.621,166.667,51.237,159.338
C00666=1020.847,-0.524,398.607,166.669,51.232,159.338
C00667=1020.852,-0.275,398.594,166.672,51.227,159.337
C00668=1020.858,-0.025,398.580,166.675,51.223,159.337
C00669=1020.864,0.225,398.565,166.678,51.217,159.337
C00670=1020.870,0.474,398.551,166.680,51.212,159.336
C00671=1020.875,0.723,398.537,166.682,51.208,159.336
C00672=1020.881,0.973,398.524,166.686,51.202,159.335
C00673=1020.887,1.222,398.510,166.688,51.198,159.335
C00674=1020.892,1.472,398.496,166.691,51.193,159.335
C00675=1020.898,1.721,398.482,166.694,51.188,159.334
C00676=1020.904,1.972,398.468,166.697,51.183,159.334
C00677=1020.910,2.220,398.454,166.699,51.178,159.333
C00678=1020.916,2.470,398.440,166.702,51.173,159.333
C00679=1020.921,2.720,398.426,166.704,51.168,159.332
C00680=1020.927,2.969,398.412,166.707,51.163,159.332
C00681=1020.933,3.219,398.398,166.710,51.158,159.331
C00682=1020.938,3.469,398.384,166.713,51.154,159.331
C00683=1020.945,3.718,398.370,166.715,51.149,159.331
C00684=1020.950,3.967,398.356,166.719,51.143,159.330
C00685=1020.956,4.217,398.343,166.721,51.139,159.330
C00686=1020.962,4.467,398.328,166.724,51.133,159.329
C00687=1020.968,4.716,398.314,166.726,51.129,159.329
C00688=1020.973,4.966,398.300,166.729,51.123,159.328
C00689=1020.979,5.215,398.286,166.732,51.119,159.328
C00690=1020.985,5.465,398.272,166.735,51.113,159.327
C00691=1020.991,5.715,398.259,166.737,51.109,159.327
C00692=1020.997,5.964,398.244,166.740,51.103,159.326
C00693=1021.002,6.213,398.230,166.742,51.098,159.326
C00694=1021.008,6.463,398.216,166.746,51.093,159.326
C00695=1021.014,6.712,398.201,166.748,51.088,159.325
C00696=1021.020,6.962,398.188,166.751,51.083,159.325
C00697=1021.026,7.211,398.174,166.753,51.078,159.324
C00698=1021.032,7.462,398.160,166.756,51.073,159.324
C00699=1021.038,7.710,398.145,166.758,51.068,159.323
C00700=1021.043,7.960,398.131,166.762,51.063,159.323
C00701=1021.048,8.210,398.118,166.764,51.058,159.322
C00702=1021.056,8.459,398.103,166.767,51.053,159.322
C00703=1021.061,8.709,398.089,166.769,51.048,159.321
C00704=1021.067,8.958,398.076,166.772,51.043,159.321
C00705=1021.073,9.208,398.061,166.775,51.038,159.320
C00706=1021.078,9.457,398.047,166.778,51.033,159.320
C00707=1021.084,9.707,398.033,166.780,51.028,159.319
C00708=1021.090,9.957,398.018,166.783,51.023,159.319
C00709=1021.096,10.206,398.005,166.786,51.018,159.319
C00710=1021.102,10.455,397.990,166.789,51.013,159.318
C00711=1021.109,10.738,397.974,166.791,51.007,159.318
C00712=1021.115,11.020,397.958,166.794,51.001,159.317
C00713=1021.122,11.304,397.942,166.798,50.996,159.317
C00714=1021.129,11.587,397.926,166.801,50.990,159.316
C00715=1021.135,11.836,397.911,166.804,50.985,159.316
C00716=1021.140,12.085,397.897,166.807,50.980,159.315
C00717=1021.147,12.334,397.883,166.809,50.975,159.315
C00718=1021.153,12.584,397.869,166.812,50.969,159.314
C00719=1021.159,12.834,397.855,166.814,50.964,159.313
C00720=1021.164,13.083,397.840,166.817,50.959,159.313
C00721=1021.170,13.333,397.826,166.819,50.954,159.313
C00722=1021.176,13.582,397.811,166.823,50.949,159.312
C00723=1021.182,13.832,397.798,166.825,50.944,159.312
C00724=1021.188,14.081,397.783,166.828,50.939,159.311
C00725=1021.194,14.331,397.768,166.830,50.934,159.311
C00726=1021.199,14.580,397.754,166.833,50.929,159.310
C00727=1021.205,14.830,397.739,166.836,50.924,159.310
C00728=1021.211,15.080,397.725,166.839,50.919,159.309
C00729=1021.216,15.329,397.710,166.841,50.914,159.309
C00730=1021.223,15.578,397.695,166.844,50.909,159.308
C00731=1021.228,15.828,397.681,166.846,50.904,159.308
C00732=1021.235,16.078,397.666,166.849,50.900,159.307
C00733=1021.240,16.327,397.652,166.852,50.894,159.307
C00734=1021.245,16.576,397.637,166.854,50.890,159.306
C00735=1021.252,16.826,397.622,166.857,50.884,159.306
C00736=1021.257,17.075,397.608,166.860,50.880,159.305
C00737=1021.263,17.325,397.594,166.863,50.874,159.305
C00738=1021.269,17.574,397.579,166.865,50.870,159.305
C00739=1021.276,17.824,397.564,166.868,50.864,159.304
C00740=1021.280,18.074,397.550,166.870,50.860,159.304
C00741=1021.286,18.323,397.535,166.874,50.854,159.303
C00742=1021.292,18.572,397.520,166.876,50.850,159.303
C00743=1021.298,18.821,397.506,166.879,50.844,159.302
C00744=1021.304,19.072,397.491,166.881,50.840,159.302
C00745=1021.310,19.321,397.477,166.884,50.834,159.301
C00746=1021.316,19.571,397.461,166.887,50.830,159.301
C00747=1021.321,19.820,397.447,166.889,50.825,159.300
C00748=1021.328,20.070,397.432,166.892,50.820,159.300
C00749=1021.333,20.319,397.417,166.894,50.815,159.299
C00750=1021.339,20.569,397.402,166.898,50.810,159.299
C00751=1021.345,20.818,397.388,166.900,50.805,159.298
C00752=1021.351,21.067,397.373,166.903,50.800,159.298
C00753=1021.356,21.317,397.358,166.905,50.795,159.297
C00754=1021.362,21.567,397.343,166.908,50.790,159.297
C00755=1021.368,21.816,397.329,166.911,50.785,159.297
C00756=1021.374,22.066,397.313,166.913,50.780,159.296
C00757=1021.379,22.315,397.299,166.916,50.775,159.296
C00758=1021.386,22.564,397.284,166.918,50.770,159.295
C00759=1021.391,22.814,397.269,166.922,50.765,159.295
C00760=1021.397,23.063,397.254,166.924,50.760,159.294
C00761=1021.403,23.313,397.240,166.927,50.754,159.294
C00762=1021.409,23.563,397.225,166.929,50.750,159.293
C00763=1021.414,23.812,397.210,166.932,50.744,159.293
C00764=1021.421,24.062,397.195,166.934,50.740,159.292
C00765=1021.426,24.311,397.180,166.937,50.734,159.292
C00766=1021.432,24.560,397.165,166.940,50.730,159.291
C00767=1021.438,24.809,397.150,166.942,50.725,159.291
C00768=1021.444,25.059,397.135,166.945,50.720,159.290
C00769=1021.450,25.309,397.119,166.947,50.715,159.290
C00770=1021.456,25.558,397.105,166.951,50.710,159.289
C00771=1021.462,25.808,397.090,166.953,50.705,159.289
C00772=1021.467,26.057,397.075,166.956,50.699,159.288
C00773=1021.473,26.307,397.060,166.958,50.694,159.288
C00774=1021.478,26.556,397.045,166.961,50.689,159.287
C00775=1021.486,26.840,397.028,166.964,50.683,159.287
C00776=1021.492,27.124,397.011,166.967,50.678,159.286
C00777=1021.499,27.408,396.994,166.970,50.672,159.286
C00778=1021.506,27.692,396.977,166.973,50.667,159.285
C00779=1021.511,27.942,396.961,166.975,50.662,159.284
C00780=1021.518,28.192,396.946,166.978,50.657,159.284
C00781=1021.523,28.441,396.931,166.981,50.652,159.283
C00782=1021.528,28.691,396.916,166.984,50.647,159.283
C00783=1021.534,28.940,396.901,166.986,50.642,159.283
C00784=1021.540,29.190,396.885,166.988,50.637,159.282
C00785=1021.547,29.439,396.870,166.992,50.632,159.282
C00786=1021.552,29.688,396.855,166.994,50.627,159.281
C00787=1021.558,29.938,396.840,166.997,50.622,159.281
C00788=1021.564,30.188,396.824,166.999,50.617,159.280
C00789=1021.569,30.437,396.810,167.003,50.612,159.280
C00790=1021.575,30.687,396.794,167.005,50.607,159.279
C00791=1021.580,30.935,396.778,167.007,50.602,159.278
C00792=1021.587,31.185,396.763,167.010,50.597,159.278
C00793=1021.592,31.435,396.748,167.012,50.592,159.278
C00794=1021.598,31.684,396.733,167.015,50.587,159.277
C00795=1021.604,31.934,396.717,167.018,50.582,159.277
C00796=1021.611,32.183,396.702,167.021,50.577,159.276
C00797=1021.616,32.432,396.687,167.023,50.572,159.276
C00798=1021.621,32.682,396.671,167.025,50.567,159.275
C00799=1021.628,32.932,396.656,167.029,50.562,159.275
C00800=1021.633,33.181,396.640,167.031,50.557,159.274
C00801=1021.639,33.430,396.625,167.034,50.552,159.274
C00802=1021.645,33.680,396.610,167.036,50.547,159.273
C00803=1021.651,33.929,396.595,167.039,50.542,159.273
C00804=1021.657,34.178,396.579,167.041,50.537,159.272
C00805=1021.663,34.428,396.564,167.044,50.532,159.272
C00806=1021.668,34.677,396.549,167.047,50.527,159.271
C00807=1021.674,34.927,396.533,167.049,50.522,159.271
C00808=1021.681,35.176,396.518,167.052,50.516,159.270
C00809=1021.686,35.426,396.502,167.054,50.512,159.269
C00810=1021.692,35.675,396.487,167.057,50.506,159.269
C00811=1021.698,35.925,396.471,167.060,50.502,159.269
C00812=1021.704,36.175,396.456,167.063,50.497,159.268
C00813=1021.710,36.424,396.441,167.065,50.491,159.267
C00814=1021.715,36.673,396.425,167.068,50.486,159.267
C00815=1021.721,36.936,396.409,167.070,50.481,159.266
C00816=1021.727,37.198,396.393,167.074,50.476,159.266
C00817=1021.734,37.461,396.376,167.075,50.471,159.265
C00818=1021.740,37.723,396.360,167.079,50.465,159.265
C00819=1021.746,37.973,396.344,167.081,50.461,159.264
C00820=1021.751,38.222,396.328,167.084,50.456,159.264
C00821=1021.757,38.472,396.312,167.086,50.451,159.263
C00822=1021.762,38.721,396.297,167.090,50.446,159.263
C00823=1021.768,38.970,396.281,167.092,50.441,159.262
C00824=1021.775,39.220,396.266,167.094,50.436,159.262
C00825=1021.781,39.469,396.249,167.097,50.430,159.261
C00826=1021.786,39.719,396.234,167.099,50.426,159.261
C00827=1021.792,39.968,396.218,167.103,50.420,159.260
C00828=1021.797,40.218,396.202,167.105,50.416,159.260
C00829=1021.804,40.467,396.187,167.107,50.411,159.259
C00830=1021.809,40.716,396.171,167.110,50.406,159.259
C00831=1021.815,40.966,396.155,167.113,50.401,159.258
C00832=1021.821,41.216,396.140,167.116,50.396,159.258
C00833=1021.827,41.465,396.123,167.118,50.390,159.257
C00834=1021.832,41.715,396.108,167.120,50.386,159.257
C00835=1021.838,41.963,396.093,167.123,50.381,159.256
C00836=1021.844,42.213,396.077,167.125,50.376,159.256
C00837=1021.850,42.463,396.061,167.129,50.371,159.255
C00838=1021.856,42.712,396.045,167.131,50.366,159.255
C00839=1021.862,42.983,396.027,167.134,50.360,159.254
C00840=1021.868,43.254,396.010,167.136,50.355,159.254
C00841=1021.874,43.526,395.993,167.139,50.350,159.253
C00842=1021.880,43.796,395.975,167.142,50.345,159.253
C00843=1021.886,44.046,395.959,167.145,50.340,159.252
C00844=1021.892,44.296,395.943,167.148,50.335,159.252
C00845=1021.897,44.544,395.927,167.150,50.330,159.251
C00846=1021.903,44.794,395.911,167.152,50.325,159.251
C00847=1021.909,45.044,395.895,167.156,50.320,159.250
C00848=1021.915,45.293,395.879,167.158,50.315,159.250
C00849=1021.921,45.542,395.863,167.160,50.310,159.249
C00850=1021.926,45.792,395.846,167.163,50.305,159.249
C00851=1021.931,46.041,395.831,167.166,50.301,159.248
C00852=1021.937,46.291,395.814,167.168,50.296,159.248
C00853=1021.943,46.540,395.798,167.171,50.291,159.247
C00854=1021.949,46.789,395.782,167.173,50.286,159.247
C00855=1021.955,47.039,395.766,167.176,50.281,159.246
C00856=1021.960,47.289,395.750,167.179,50.276,159.246
C00857=1021.966,47.538,395.734,167.181,50.271,159.245
C00858=1021.971,47.787,395.717,167.183,50.266,159.244
C00859=1021.977,48.036,395.701,167.186,50.261,159.244
C00860=1021.983,48.286,395.685,167.189,50.256,159.243
C00861=1021.988,48.536,395.669,167.192,50.251,159.243
C00862=1021.994,48.785,395.653,167.194,50.246,159.243
C00863=1022.000,49.034,395.637,167.196,50.242,159.242
C00864=1022.006,49.284,395.621,167.200,50.236,159.242
C00865=1022.012,49.533,395.604,167.202,50.232,159.241
C00866=1022.018,49.782,395.588,167.204,50.226,159.240
C00867=1022.023,50.032,395.571,167.207,50.221,159.240
C00868=1022.029,50.281,395.555,167.209,50.216,159.239
C00869=1022.034,50.531,395.540,167.213,50.211,159.239
C00870=1022.040,50.780,395.523,167.215,50.207,159.238
C00871=1022.046,51.029,395.507,167.217,50.202,159.238
C00872=1022.052,51.279,395.491,167.221,50.197,159.237
C00873=1022.058,51.528,395.475,167.222,50.191,159.237
C00874=1022.064,51.777,395.458,167.225,50.187,159.236
C00875=1022.069,52.027,395.442,167.228,50.182,159.236
C00876=1022.075,52.276,395.425,167.230,50.177,159.235
C00877=1022.081,52.526,395.409,167.234,50.172,159.235
C00878=1022.087,52.775,395.393,167.236,50.167,159.234
C00879=1022.093,53.024,395.377,167.238,50.161,159.234
C00880=1022.099,53.274,395.360,167.241,50.156,159.233
C00881=1022.105,53.523,395.344,167.243,50.152,159.233
C00882=1022.110,53.773,395.327,167.247,50.147,159.232
C00883=1022.116,54.023,395.312,167.248,50.141,159.231
C00884=1022.122,54.272,395.295,167.252,50.136,159.231
C00885=1022.128,54.521,395.279,167.254,50.131,159.230
C00886=1022.134,54.771,395.263,167.256,50.127,159.230
C00887=1022.140,55.020,395.247,167.260,50.122,159.229
C00888=1022.146,55.269,395.230,167.261,50.116,159.229
C00889=1022.151,55.519,395.214,167.265,50.111,159.228
C00890=1022.157,55.769,395.197,167.267,50.106,159.228
C00891=1022.163,56.018,395.181,167.269,50.102,159.227
C00892=1022.169,56.267,395.164,167.272,50.096,159.227
C00893=1022.175,56.516,395.148,167.275,50.091,159.226
C00894=1022.181,56.765,395.132,167.278,50.086,159.226
C00895=1022.187,57.015,395.115,167.280,50.081,159.225
C00896=1022.192,57.264,395.098,167.283,50.076,159.225
C00897=1022.198,57.514,395.082,167.285,50.071,159.224
C00898=1022.204,57.763,395.066,167.288,50.066,159.223
C00899=1022.210,58.012,395.050,167.290,50.060,159.223
C00900=1022.216,58.262,395.033,167.293,50.056,159.222
C00901=1022.222,58.511,395.017,167.296,50.051,159.222
C00902=1022.228,58.760,395.001,167.298,50.045,159.221
C00903=1022.234,59.045,394.982,167.301,50.039,159.221
C00904=1022.241,59.328,394.963,167.304,50.034,159.220
C00905=1022.248,59.612,394.944,167.307,50.028,159.219
C00906=1022.254,59.897,394.926,167.311,50.022,159.219
C00907=1022.260,60.145,394.909,167.313,50.017,159.218
C00908=1022.266,60.395,394.892,167.315,50.012,159.218
C00909=1022.273,60.645,394.876,167.318,50.007,159.217
C00910=1022.279,60.894,394.860,167.321,50.002,159.217
C00911=1022.285,61.143,394.843,167.323,49.996,159.216
C00912=1022.290,61.393,394.826,167.326,49.991,159.215
C00913=1022.296,61.642,394.810,167.329,49.986,159.215
C00914=1022.302,61.891,394.793,167.331,49.981,159.214
C00915=1022.308,62.140,394.777,167.334,49.976,159.214
C00916=1022.314,62.390,394.761,167.336,49.970,159.213
C00917=1022.320,62.639,394.744,167.340,49.965,159.213
C00918=1022.326,62.889,394.727,167.342,49.961,159.212
C00919=1022.332,63.138,394.710,167.345,49.955,159.211
C00920=1022.338,63.388,394.694,167.347,49.950,159.211
C00921=1022.343,63.637,394.677,167.349,49.945,159.210
C00922=1022.349,63.887,394.661,167.353,49.940,159.210
C00923=1022.355,64.136,394.643,167.355,49.936,159.209
C00924=1022.361,64.386,394.627,167.358,49.930,159.209
C00925=1022.367,64.635,394.609,167.360,49.925,159.208
C00926=1022.373,64.884,394.593,167.362,49.921,159.208
C00927=1022.378,65.134,394.576,167.366,49.916,159.207
C00928=1022.384,65.382,394.559,167.368,49.910,159.207
C00929=1022.390,65.632,394.543,167.371,49.905,159.206
C00930=1022.396,65.881,394.526,167.373,49.900,159.206
C00931=1022.402,66.131,394.509,167.376,49.896,159.205
C00932=1022.408,66.381,394.492,167.379,49.890,159.204
C00933=1022.414,66.629,394.475,167.381,49.885,159.204
C00934=1022.419,66.879,394.458,167.384,49.880,159.204
C00935=1022.425,67.128,394.440,167.386,49.875,159.203
C00936=1022.431,67.377,394.424,167.388,49.870,159.202
C00937=1022.436,67.628,394.407,167.392,49.865,159.202
C00938=1022.443,67.876,394.390,167.394,49.860,159.201
C00939=1022.448,68.126,394.373,167.397,49.855,159.201
C00940=1022.454,68.375,394.356,167.399,49.850,159.200
C00941=1022.459,68.624,394.339,167.402,49.845,159.200
C00942=1022.466,68.874,394.322,167.405,49.840,159.199
C00943=1022.471,69.124,394.305,167.407,49.835,159.199
C00944=1022.477,69.373,394.288,167.409,49.831,159.198
C00945=1022.483,69.622,394.271,167.412,49.825,159.197
C00946=1022.488,69.871,394.254,167.415,49.820,159.197
C00947=1022.494,70.121,394.236,167.418,49.815,159.196
C00948=1022.500,70.370,394.220,167.420,49.811,159.196
C00949=1022.506,70.619,394.202,167.422,49.805,159.195
C00950=1022.511,70.869,394.185,167.426,49.800,159.195
C00951=1022.517,71.117,394.168,167.428,49.795,159.194
C00952=1022.524,71.367,394.150,167.431,49.790,159.194
C00953=1022.529,71.617,394.133,167.434,49.786,159.193
C00954=1022.535,71.866,394.116,167.436,49.780,159.193
C00955=1022.540,72.115,394.100,167.439,49.775,159.192
C00956=1022.546,72.365,394.082,167.441,49.771,159.192
C00957=1022.553,72.614,394.065,167.443,49.766,159.191
C00958=1022.558,72.863,394.048,167.446,49.760,159.190
C00959=1022.563,73.112,394.030,167.449,49.755,159.190
C00960=1022.569,73.362,394.012,167.452,49.750,159.189
C00961=1022.575,73.612,393.996,167.454,49.746,159.189
C00962=1022.581,73.861,393.978,167.456,49.740,159.188
C00963=1022.586,74.110,393.961,167.460,49.735,159.188
C00964=1022.593,74.360,393.944,167.462,49.731,159.187
C00965=1022.598,74.609,393.927,167.465,49.726,159.187
C00966=1022.604,74.858,393.909,167.467,49.720,159.186
C00967=1022.611,75.141,393.890,167.470,49.715,159.185
C00968=1022.617,75.426,393.869,167.473,49.709,159.185
C00969=1022.624,75.709,393.850,167.476,49.703,159.184
C00970=1022.631,75.993,393.831,167.479,49.697,159.184
C00971=1022.637,76.242,393.813,167.482,49.692,159.183
C00972=1022.643,76.492,393.795,167.485,49.688,159.183
C00973=1022.648,76.741,393.778,167.487,49.683,159.182
C00974=1022.653,76.991,393.761,167.490,49.677,159.181
C00975=1022.659,77.240,393.743,167.492,49.673,159.181
C00976=1022.666,77.489,393.726,167.495,49.668,159.180
C00977=1022.671,77.738,393.708,167.498,49.663,159.180
C00978=1022.677,77.987,393.691,167.500,49.658,159.179
C00979=1022.683,78.237,393.674,167.503,49.653,159.179
C00980=1022.688,78.486,393.656,167.506,49.648,159.178
C00981=1022.694,78.735,393.638,167.508,49.643,159.178
C00982=1022.700,78.985,393.621,167.511,49.638,159.177
C00983=1022.705,79.234,393.603,167.514,49.634,159.177
C00984=1022.711,79.483,393.585,167.516,49.628,159.176
C00985=1022.717,79.733,393.567,167.519,49.623,159.176
C00986=1022.723,79.982,393.550,167.521,49.618,159.175
C00987=1022.728,80.231,393.532,167.524,49.614,159.174
C00988=1022.734,80.481,393.514,167.527,49.609,159.174
C00989=1022.740,80.730,393.497,167.529,49.603,159.173
C00990=1022.745,80.979,393.479,167.532,49.598,159.173
C00991=1022.751,81.229,393.461,167.535,49.594,159.172
C00992=1022.757,81.478,393.444,167.537,49.589,159.172
C00993=1022.762,81.727,393.426,167.540,49.584,159.171
C00994=1022.768,81.977,393.408,167.542,49.579,159.171
C00995=1022.774,82.226,393.391,167.545,49.574,159.170
C00996=1022.780,82.475,393.373,167.548,49.569,159.170
C00997=1022.786,82.724,393.355,167.550,49.564,159.169
C00998=1022.791,82.973,393.338,167.553,49.559,159.168
C00999=1022.797,83.223,393.320,167.556,49.554,159.168
C01000=1022.803,83.472,393.302,167.558,49.549,159.167
C01001=1022.809,83.722,393.284,167.561,49.544,159.167
C01002=1022.814,83.971,393.267,167.563,49.539,159.166
C01003=1022.820,84.220,393.249,167.567,49.534,159.166
C01004=1022.826,84.470,393.231,167.569,49.529,159.165
C01005=1022.832,84.719,393.214,167.571,49.525,159.165
C01006=1022.838,84.969,393.196,167.574,49.519,159.164
C01007=1022.843,85.218,393.178,167.576,49.514,159.163
C01008=1022.849,85.467,393.160,167.580,49.509,159.163
C01009=1022.855,85.716,393.143,167.582,49.504,159.162
C01010=1022.860,85.965,393.125,167.585,49.499,159.162
C01011=1022.867,86.215,393.107,167.587,49.494,159.161
C01012=1022.872,86.464,393.090,167.590,49.490,159.161
C01013=1022.878,86.713,393.071,167.593,49.484,159.160
C01014=1022.884,86.962,393.053,167.595,49.479,159.160
C01015=1022.890,87.212,393.035,167.599,49.474,159.159
C01016=1022.896,87.461,393.018,167.600,49.469,159.158
C01017=1022.902,87.711,393.000,167.604,49.464,159.158
C01018=1022.907,87.960,392.982,167.606,49.459,159.157
C01019=1022.913,88.210,392.964,167.608,49.454,159.157
C01020=1022.919,88.458,392.946,167.612,49.449,159.156
C01021=1022.925,88.708,392.928,167.614,49.444,159.156
C01022=1022.931,88.957,392.911,167.617,49.439,159.155
C01023=1022.937,89.207,392.893,167.619,49.434,159.155
C01024=1022.942,89.456,392.874,167.623,49.429,159.154
C01025=1022.948,89.705,392.856,167.625,49.424,159.154
C01026=1022.954,89.954,392.838,167.627,49.419,159.153
C01027=1022.959,90.204,392.820,167.630,49.414,159.152
C01028=1022.965,90.453,392.802,167.633,49.409,159.152
C01029=1022.971,90.702,392.784,167.635,49.405,159.151
C01030=1022.976,90.952,392.765,167.638,49.400,159.151
C01031=1022.982,91.235,392.745,167.641,49.394,159.150
C01032=1022.989,91.519,392.724,167.644,49.388,159.150
C01033=1022.995,91.803,392.704,167.647,49.383,159.149
C01034=1023.002,92.087,392.683,167.650,49.377,159.148
C01035=1023.008,92.335,392.664,167.653,49.372,159.148
C01036=1023.013,92.585,392.646,167.656,49.367,159.147
C01037=1023.019,92.834,392.628,167.658,49.362,159.147
C01038=1023.025,93.083,392.610,167.660,49.357,159.146
C01039=1023.030,93.333,392.592,167.664,49.352,159.146
C01040=1023.036,93.582,392.574,167.666,49.348,159.145
C01041=1023.042,93.831,392.555,167.669,49.342,159.145
C01042=1023.047,94.081,392.537,167.671,49.338,159.144
C01043=1023.054,94.330,392.518,167.674,49.333,159.143
C01044=1023.059,94.579,392.501,167.677,49.328,159.143
C01045=1023.065,94.828,392.481,167.679,49.323,159.142
C01046=1023.071,95.078,392.464,167.683,49.318,159.142
C01047=1023.077,95.327,392.446,167.685,49.313,159.141
C01048=1023.082,95.576,392.427,167.687,49.308,159.141
C01049=1023.088,95.826,392.409,167.690,49.303,159.140
C01050=1023.094,96.074,392.391,167.693,49.298,159.140
C01051=1023.099,96.324,392.372,167.696,49.293,159.139
C01052=1023.106,96.573,392.354,167.698,49.288,159.139
C01053=1023.111,96.822,392.336,167.701,49.283,159.138
C01054=1023.117,97.072,392.317,167.704,49.278,159.137
C01055=1023.122,97.321,392.299,167.706,49.273,159.137
C01056=1023.129,97.570,392.281,167.709,49.268,159.136
C01057=1023.134,97.820,392.262,167.711,49.263,159.136
C01058=1023.140,98.068,392.244,167.715,49.258,159.135
C01059=1023.146,98.318,392.226,167.717,49.254,159.135
C01060=1023.151,98.567,392.207,167.720,49.248,159.134
C01061=1023.157,98.817,392.189,167.723,49.243,159.134
C01062=1023.164,99.066,392.170,167.726,49.238,159.133
C01063=1023.168,99.315,392.152,167.728,49.233,159.132
C01064=1023.175,99.564,392.134,167.731,49.228,159.132
C01065=1023.181,99.814,392.114,167.734,49.223,159.131
C01066=1023.186,100.063,392.097,167.736,49.219,159.131
C01067=1023.192,100.312,392.078,167.739,49.214,159.130
C01068=1023.197,100.562,392.058,167.741,49.209,159.130
C01069=1023.203,100.811,392.041,167.744,49.204,159.129
C01070=1023.209,101.060,392.021,167.747,49.199,159.129
C01071=1023.215,101.308,392.003,167.750,49.194,159.128
C01072=1023.220,101.558,391.984,167.753,49.189,159.128
C01073=1023.226,101.808,391.965,167.755,49.185,159.127
C01074=1023.231,102.056,391.947,167.757,49.179,159.126
C01075=1023.237,102.306,391.928,167.761,49.175,159.126
C01076=1023.242,102.556,391.909,167.763,49.170,159.125
C01077=1023.248,102.804,391.891,167.766,49.165,159.125
C01078=1023.254,103.054,391.872,167.769,49.160,159.124
C01079=1023.260,103.303,391.853,167.771,49.155,159.124
C01080=1023.266,103.552,391.834,167.774,49.150,159.123
C01081=1023.271,103.802,391.816,167.777,49.145,159.123
C01082=1023.277,104.051,391.797,167.780,49.141,159.122
C01083=1023.282,104.299,391.778,167.782,49.136,159.122
C01084=1023.288,104.549,391.759,167.785,49.130,159.121
C01085=1023.294,104.799,391.741,167.788,49.126,159.121
C01086=1023.300,105.048,391.722,167.790,49.121,159.120
C01087=1023.306,105.297,391.704,167.794,49.116,159.120
C01088=1023.311,105.546,391.684,167.796,49.111,159.119
C01089=1023.317,105.795,391.665,167.799,49.106,159.118
C01090=1023.323,106.044,391.647,167.801,49.101,159.118
C01091=1023.328,106.294,391.628,167.805,49.096,159.117
C01092=1023.334,106.543,391.609,167.807,49.091,159.117
C01093=1023.340,106.792,391.590,167.810,49.086,159.116
C01094=1023.346,107.041,391.571,167.812,49.081,159.116
C01095=1023.352,107.325,391.550,167.816,49.076,159.115
C01096=1023.359,107.609,391.528,167.819,49.070,159.114
C01097=1023.365,107.893,391.507,167.822,49.065,159.114
C01098=1023.372,108.177,391.486,167.825,49.059,159.113
C01099=1023.377,108.426,391.467,167.828,49.054,159.113
C01100=1023.384,108.675,391.448,167.830,49.049,159.112
C01101=1023.389,108.924,391.429,167.834,49.044,159.111
C01102=1023.395,109.174,391.410,167.836,49.039,159.111
C01103=1023.401,109.422,391.391,167.839,49.034,159.110
C01104=1023.407,109.672,391.372,167.841,49.029,159.110
C01105=1023.412,109.921,391.353,167.845,49.024,159.109
C01106=1023.418,110.170,391.333,167.847,49.019,159.109
C01107=1023.424,110.420,391.315,167.851,49.015,159.108
C01108=1023.430,110.668,391.296,167.853,49.009,159.108
C01109=1023.435,110.918,391.277,167.856,49.004,159.107
C01110=1023.441,111.167,391.257,167.858,49.000,159.107
C01111=1023.447,111.417,391.238,167.861,48.995,159.106
C01112=1023.452,111.665,391.219,167.864,48.990,159.106
C01113=1023.458,111.914,391.201,167.866,48.985,159.105
C01114=1023.464,112.164,391.181,167.870,48.980,159.104
C01115=1023.470,112.413,391.162,167.872,48.975,159.104
C01116=1023.475,112.663,391.143,167.875,48.971,159.103
C01117=1023.481,112.912,391.124,167.878,48.966,159.103
C01118=1023.486,113.161,391.105,167.880,48.961,159.102
C01119=1023.492,113.410,391.085,167.884,48.956,159.102
C01120=1023.498,113.659,391.066,167.886,48.952,159.101
C01121=1023.503,113.909,391.046,167.889,48.947,159.101
C01122=1023.508,114.158,391.027,167.891,48.942,159.100
C01123=1023.513,114.407,391.008,167.894,48.937,159.100
C01124=1023.519,114.656,390.988,167.897,48.932,159.099
C01125=1023.525,114.905,390.968,167.900,48.927,159.099
C01126=1023.531,115.155,390.949,167.903,48.923,159.098
C01127=1023.537,115.404,390.929,167.905,48.918,159.098
C01128=1023.542,115.652,390.910,167.909,48.913,159.097
C01129=1023.548,115.902,390.891,167.911,48.908,159.097
C01130=1023.553,116.151,390.872,167.914,48.904,159.096
C01131=1023.558,116.400,390.851,167.917,48.899,159.096
C01132=1023.564,116.650,390.832,167.919,48.894,159.095
C01133=1023.570,116.899,390.813,167.922,48.889,159.094
C01134=1023.576,117.148,390.793,167.925,48.884,159.094
C01135=1023.581,117.397,390.774,167.928,48.879,159.093
C01136=1023.587,117.646,390.755,167.931,48.875,159.093
C01137=1023.593,117.895,390.735,167.933,48.870,159.092
C01138=1023.598,118.144,390.716,167.936,48.865,159.092
C01139=1023.603,118.394,390.696,167.939,48.861,159.091
C01140=1023.609,118.643,390.676,167.942,48.856,159.091
C01141=1023.615,118.892,390.657,167.945,48.851,159.090
C01142=1023.621,119.142,390.637,167.948,48.846,159.090
C01143=1023.626,119.390,390.618,167.950,48.841,159.089
C01144=1023.632,119.639,390.598,167.953,48.836,159.089
C01145=1023.637,119.889,390.579,167.956,48.831,159.088
C01146=1023.643,120.138,390.559,167.959,48.827,159.088
C01147=1023.648,120.387,390.539,167.962,48.822,159.087
C01148=1023.654,120.636,390.519,167.965,48.817,159.087
C01149=1023.660,120.886,390.500,167.967,48.812,159.086
C01150=1023.666,121.135,390.481,167.971,48.807,159.085
C01151=1023.672,121.384,390.461,167.973,48.802,159.085
C01152=1023.677,121.633,390.442,167.976,48.797,159.084
C01153=1023.683,121.882,390.422,167.979,48.793,159.084
C01154=1023.689,122.131,390.403,167.982,48.788,159.083
C01155=1023.694,122.381,390.382,167.984,48.783,159.083
C01156=1023.700,122.630,390.363,167.988,48.778,159.082
C01157=1023.706,122.879,390.343,167.990,48.773,159.082
C01158=1023.711,123.128,390.324,167.994,48.768,159.081
C01159=1023.718,123.412,390.301,167.997,48.763,159.081
C01160=1023.725,123.696,390.279,168.000,48.757,159.080
C01161=1023.731,123.979,390.257,168.003,48.752,159.079
C01162=1023.738,124.263,390.234,168.006,48.746,159.079
C01163=1023.743,124.512,390.214,168.009,48.741,159.078
C01164=1023.749,124.761,390.194,168.012,48.737,159.078
C01165=1023.755,125.010,390.175,168.015,48.732,159.077
C01166=1023.760,125.260,390.155,168.018,48.727,159.077
C01167=1023.766,125.509,390.135,168.021,48.722,159.076
C01168=1023.772,125.758,390.116,168.023,48.717,159.075
C01169=1023.778,126.007,390.096,168.026,48.712,159.075
C01170=1023.783,126.257,390.076,168.029,48.708,159.074
C01171=1023.789,126.505,390.056,168.032,48.703,159.074
C01172=1023.795,126.755,390.037,168.035,48.697,159.073
C01173=1023.801,127.004,390.017,168.038,48.693,159.073
C01174=1023.807,127.252,389.997,168.041,48.688,159.072
C01175=1023.812,127.502,389.978,168.044,48.683,159.072
C01176=1023.818,127.751,389.958,168.047,48.678,159.071
C01177=1023.823,128.000,389.938,168.049,48.673,159.071
C01178=1023.829,128.249,389.918,168.053,48.668,159.070
C01179=1023.835,128.498,389.898,168.055,48.664,159.070
C01180=1023.841,128.747,389.879,168.058,48.659,159.069
C01181=1023.848,128.997,389.859,168.062,48.653,159.068
C01182=1023.854,129.246,389.839,168.064,48.649,159.068
C01183=1023.859,129.496,389.819,168.067,48.644,159.067
C01184=1023.865,129.744,389.799,168.070,48.639,159.067
C01185=1023.871,129.993,389.779,168.073,48.634,159.066
C01186=1023.876,130.243,389.760,168.076,48.629,159.066
C01187=1023.882,130.492,389.739,168.079,48.624,159.065
C01188=1023.888,130.740,389.719,168.082,48.619,159.065
C01189=1023.893,130.990,389.699,168.085,48.615,159.064
C01190=1023.899,131.238,389.679,168.088,48.610,159.064
C01191=1023.904,131.488,389.659,168.090,48.605,159.063
C01192=1023.910,131.737,389.639,168.094,48.601,159.063
C01193=1023.916,131.987,389.618,168.096,48.596,159.062
C01194=1023.922,132.236,389.598,168.100,48.591,159.062
C01195=1023.927,132.485,389.577,168.102,48.587,159.061
C01196=1023.933,132.734,389.557,168.106,48.582,159.061
C01197=1023.938,132.983,389.537,168.108,48.577,159.060
C01198=1023.944,133.232,389.518,168.111,48.572,159.059
C01199=1023.949,133.481,389.497,168.114,48.567,159.059
C01200=1023.955,133.730,389.477,168.117,48.562,159.058
C01201=1023.960,133.979,389.457,168.120,48.557,159.058
C01202=1023.967,134.229,389.436,168.123,48.553,159.057
C01203=1023.972,134.478,389.416,168.126,48.548,159.057
C01204=1023.978,134.727,389.396,168.129,48.543,159.056
C01205=1023.983,134.976,389.375,168.132,48.539,159.056
C01206=1023.989,135.225,389.355,168.135,48.534,159.055
C01207=1023.995,135.474,389.335,168.138,48.529,159.055
C01208=1024.001,135.722,389.315,168.140,48.525,159.054
C01209=1024.006,135.972,389.294,168.144,48.519,159.054
C01210=1024.012,136.221,389.274,168.147,48.514,159.053
C01211=1024.018,136.470,389.253,168.149,48.510,159.053
C01212=1024.024,136.719,389.233,168.153,48.505,159.052
C01213=1024.029,136.968,389.213,168.155,48.500,159.052
C01214=1024.035,137.218,389.192,168.159,48.495,159.051
C01215=1024.041,137.467,389.172,168.161,48.491,159.051
C01216=1024.046,137.716,389.151,168.165,48.486,159.050
C01217=1024.052,137.965,389.131,168.168,48.481,159.050
C01218=1024.057,138.214,389.111,168.171,48.477,159.049
C01219=1024.064,138.463,389.091,168.174,48.472,159.049
C01220=1024.069,138.713,389.070,168.176,48.467,159.048
C01221=1024.074,138.962,389.049,168.180,48.462,159.048
C01222=1024.080,139.210,389.028,168.182,48.458,159.047
C01223=1024.086,139.494,389.005,168.186,48.452,159.047
C01224=1024.093,139.778,388.982,168.190,48.447,159.046
C01225=1024.099,140.061,388.958,168.193,48.442,159.046
C01226=1024.106,140.345,388.935,168.196,48.436,159.045
C01227=1024.111,140.594,388.914,168.200,48.431,159.044
C01228=1024.117,140.844,388.893,168.202,48.427,159.044
C01229=1024.123,141.092,388.873,168.205,48.422,159.043
C01230=1024.128,141.341,388.852,168.209,48.417,159.043
C01231=1024.134,141.591,388.831,168.211,48.413,159.042
C01232=1024.139,141.840,388.810,168.215,48.408,159.042
C01233=1024.145,142.089,388.790,168.217,48.403,159.041
C01234=1024.151,142.337,388.769,168.221,48.398,159.041
C01235=1024.157,142.587,388.748,168.223,48.394,159.040
C01236=1024.162,142.836,388.728,168.227,48.389,159.040
C01237=1024.168,143.085,388.708,168.230,48.384,159.039
C01238=1024.174,143.334,388.686,168.233,48.380,159.039
C01239=1024.179,143.583,388.666,168.236,48.375,159.038
C01240=1024.185,143.832,388.645,168.239,48.370,159.038
C01241=1024.190,144.081,388.624,168.242,48.366,159.037
C01242=1024.197,144.330,388.603,168.245,48.361,159.037
C01243=1024.202,144.579,388.583,168.248,48.356,159.036
C01244=1024.207,144.829,388.562,168.251,48.351,159.036
C01245=1024.213,145.078,388.541,168.255,48.347,159.035
C01246=1024.219,145.327,388.521,168.257,48.342,159.035
C01247=1024.225,145.575,388.499,168.261,48.337,159.034
C01248=1024.231,145.825,388.478,168.264,48.332,159.034
C01249=1024.236,146.074,388.458,168.267,48.328,159.033
C01250=1024.242,146.323,388.437,168.270,48.323,159.033
C01251=1024.248,146.572,388.416,168.272,48.318,159.032
C01252=1024.253,146.821,388.394,168.276,48.314,159.032
C01253=1024.258,147.070,388.374,168.279,48.309,159.031
C01254=1024.265,147.319,388.352,168.282,48.304,159.031
C01255=1024.270,147.568,388.332,168.285,48.300,159.030
C01256=1024.275,147.817,388.311,168.289,48.295,159.030
C01257=1024.281,148.067,388.290,168.292,48.291,159.030
C01258=1024.287,148.315,388.268,168.295,48.286,159.029
C01259=1024.293,148.564,388.248,168.297,48.282,159.028
C01260=1024.299,148.813,388.227,168.301,48.277,159.028
C01261=1024.304,149.062,388.206,168.304,48.272,159.028
C01262=1024.309,149.311,388.184,168.307,48.267,159.027
C01263=1024.315,149.561,388.163,168.310,48.263,159.027
C01264=1024.320,149.809,388.142,168.314,48.258,159.026
C01265=1024.326,150.059,388.121,168.316,48.253,159.025
C01266=1024.332,150.308,388.100,168.320,48.248,159.025
C01267=1024.337,150.556,388.079,168.322,48.245,159.025
C01268=1024.343,150.806,388.058,168.326,48.240,159.024
C01269=1024.349,151.055,388.036,168.329,48.235,159.024
C01270=1024.355,151.304,388.015,168.332,48.230,159.023
C01271=1024.360,151.553,387.994,168.335,48.226,159.023
C01272=1024.366,151.801,387.973,168.339,48.221,159.022
C01273=1024.372,152.051,387.952,168.341,48.216,159.022
C01274=1024.377,152.300,387.931,168.345,48.212,159.021
C01275=1024.383,152.549,387.909,168.348,48.207,159.021
C01276=1024.389,152.798,387.889,168.351,48.202,159.020
C01277=1024.395,153.047,387.867,168.354,48.198,159.020
C01278=1024.400,153.296,387.846,168.358,48.193,159.019
C01279=1024.406,153.545,387.823,168.360,48.189,159.019
C01280=1024.411,153.794,387.803,168.364,48.184,159.018
C01281=1024.417,154.043,387.782,168.367,48.179,159.018
C01282=1024.423,154.292,387.760,168.370,48.175,159.017
C01283=1024.428,154.541,387.739,168.373,48.170,159.017
C01284=1024.433,154.791,387.717,168.377,48.166,159.017
C01285=1024.439,155.039,387.696,168.380,48.161,159.016
C01286=1024.445,155.289,387.674,168.383,48.156,159.016
C01287=1024.452,155.571,387.650,168.386,48.151,159.015
C01288=1024.458,155.855,387.626,168.391,48.146,159.014
C01289=1024.464,156.138,387.601,168.394,48.140,159.014
C01290=1024.471,156.422,387.576,168.397,48.136,159.013
C01291=1024.476,156.671,387.556,168.401,48.131,159.013
C01292=1024.482,156.920,387.534,168.404,48.126,159.012
C01293=1024.487,157.169,387.512,168.408,48.121,159.012
C01294=1024.493,157.418,387.491,168.410,48.117,159.011
C01295=1024.499,157.667,387.469,168.414,48.113,159.011
C01296=1024.505,157.916,387.448,168.418,48.108,159.011
C01297=1024.511,158.164,387.426,168.420,48.103,159.010
C01298=1024.516,158.414,387.404,168.423,48.099,159.010
C01299=1024.522,158.662,387.383,168.427,48.094,159.009
C01300=1024.528,158.912,387.361,168.430,48.089,159.009
C01301=1024.534,159.161,387.340,168.433,48.085,159.008
C01302=1024.539,159.410,387.318,168.437,48.080,159.008
C01303=1024.544,159.659,387.296,168.440,48.076,159.007
C01304=1024.550,159.908,387.274,168.443,48.072,159.007
C01305=1024.555,160.157,387.252,168.446,48.067,159.006
C01306=1024.560,160.406,387.230,168.449,48.063,159.006
C01307=1024.566,160.655,387.209,168.453,48.059,159.006
C01308=1024.571,160.904,387.187,168.456,48.054,159.005
C01309=1024.577,161.153,387.164,168.459,48.050,159.005
C01310=1024.582,161.401,387.142,168.463,48.045,159.004
C01311=1024.588,161.651,387.120,168.466,48.040,159.004
C01312=1024.593,161.900,387.098,168.469,48.037,159.003
C01313=1024.599,162.149,387.077,168.472,48.032,159.003
C01314=1024.604,162.397,387.054,168.476,48.028,159.003
C01315=1024.609,162.647,387.032,168.479,48.023,159.002
C01316=1024.615,162.896,387.010,168.482,48.018,159.002
C01317=1024.620,163.145,386.988,168.486,48.014,159.001
C01318=1024.626,163.393,386.966,168.488,48.010,159.001
C01319=1024.632,163.642,386.944,168.492,48.006,159.000
C01320=1024.637,163.892,386.922,168.496,48.001,159.000
C01321=1024.642,164.140,386.900,168.498,47.996,158.999
C01322=1024.648,164.389,386.878,168.502,47.992,158.999
C01323=1024.654,164.638,386.856,168.505,47.988,158.999
C01324=1024.659,164.887,386.834,168.509,47.983,158.998
C01325=1024.665,165.136,386.811,168.512,47.979,158.998
C01326=1024.670,165.385,386.789,168.515,47.974,158.997
C01327=1024.675,165.634,386.767,168.519,47.970,158.997
C01328=1024.682,165.883,386.745,168.522,47.966,158.996
C01329=1024.687,166.132,386.723,168.525,47.961,158.996
C01330=1024.692,166.381,386.701,168.529,47.957,158.996
C01331=1024.698,166.630,386.678,168.532,47.952,158.995
C01332=1024.703,166.878,386.657,168.535,47.948,158.995
C01333=1024.709,167.128,386.634,168.539,47.944,158.994
C01334=1024.714,167.377,386.611,168.542,47.939,158.994
C01335=1024.720,167.625,386.590,168.546,47.935,158.993
C01336=1024.726,167.874,386.567,168.548,47.930,158.993
C01337=1024.731,168.124,386.545,168.552,47.925,158.992
C01338=1024.737,168.372,386.524,168.556,47.921,158.992
C01339=1024.742,168.621,386.501,168.559,47.917,158.992
C01340=1024.748,168.871,386.479,168.562,47.913,158.991
C01341=1024.754,169.119,386.456,168.566,47.908,158.991
C01342=1024.759,169.368,386.434,168.569,47.903,158.990
C01343=1024.765,169.617,386.411,168.573,47.899,158.990
C01344=1024.771,169.866,386.390,168.576,47.894,158.989
C01345=1024.777,170.115,386.367,168.579,47.890,158.989
C01346=1024.782,170.364,386.345,168.583,47.886,158.989
C01347=1024.787,170.613,386.322,168.586,47.881,158.988
C01348=1024.794,170.862,386.300,168.590,47.877,158.988
C01349=1024.799,171.111,386.277,168.594,47.872,158.987
C01350=1024.804,171.360,386.256,168.596,47.868,158.987
C01351=1024.811,171.643,386.230,168.601,47.863,158.986
C01352=1024.817,171.926,386.205,168.604,47.858,158.986
C01353=1024.824,172.209,386.179,168.609,47.853,158.985
C01354=1024.831,172.491,386.154,168.612,47.848,158.985
C01355=1024.836,172.741,386.131,168.616,47.844,158.985
C01356=1024.842,172.989,386.109,168.619,47.839,158.984
C01357=1024.847,173.239,386.087,168.623,47.835,158.984
C01358=1024.853,173.487,386.064,168.626,47.830,158.983
C01359=1024.859,173.736,386.041,168.630,47.825,158.983
C01360=1024.865,173.986,386.019,168.633,47.822,158.982
C01361=1024.870,174.234,385.997,168.636,47.817,158.982
C01362=1024.876,174.482,385.974,168.640,47.813,158.982
C01363=1024.882,174.732,385.952,168.644,47.808,158.981
C01364=1024.887,174.981,385.929,168.647,47.803,158.981
C01365=1024.894,175.230,385.907,168.651,47.799,158.980
C01366=1024.899,175.479,385.884,168.654,47.794,158.980
C01367=1024.905,175.728,385.861,168.658,47.790,158.980
C01368=1024.911,175.976,385.840,168.661,47.786,158.979
C01369=1024.916,176.225,385.817,168.664,47.781,158.978
C01370=1024.922,176.474,385.794,168.668,47.777,158.978
C01371=1024.928,176.723,385.771,168.672,47.772,158.978
C01372=1024.934,176.972,385.750,168.675,47.768,158.977
C01373=1024.940,177.221,385.727,168.679,47.764,158.977
C01374=1024.945,177.470,385.704,168.682,47.759,158.976
C01375=1024.951,177.719,385.681,168.686,47.755,158.976
C01376=1024.957,177.968,385.659,168.690,47.750,158.976
C01377=1024.963,178.217,385.636,168.694,47.746,158.975
C01378=1024.969,178.466,385.613,168.697,47.741,158.975
C01379=1024.974,178.715,385.590,168.701,47.737,158.974
C01380=1024.981,178.963,385.568,168.703,47.733,158.974
C01381=1024.986,179.212,385.546,168.707,47.728,158.973
C01382=1024.991,179.461,385.523,168.711,47.724,158.973
C01383=1024.998,179.710,385.501,168.714,47.719,158.973
C01384=1025.004,179.959,385.478,168.718,47.715,158.972
C01385=1025.009,180.208,385.455,168.722,47.710,158.972
C01386=1025.015,180.456,385.432,168.725,47.706,158.971
C01387=1025.021,180.706,385.410,168.729,47.702,158.971
C01388=1025.027,180.955,385.388,168.733,47.697,158.971
C01389=1025.033,181.203,385.365,168.736,47.693,158.970
C01390=1025.039,181.452,385.342,168.740,47.688,158.970
C01391=1025.045,181.701,385.319,168.743,47.684,158.969
C01392=1025.051,181.950,385.296,168.747,47.679,158.969
C01393=1025.057,182.199,385.273,168.751,47.675,158.968
C01394=1025.063,182.448,385.250,168.755,47.671,158.968
C01395=1025.069,182.697,385.227,168.758,47.666,158.968
C01396=1025.074,182.946,385.204,168.762,47.662,158.967
C01397=1025.079,183.195,385.181,168.766,47.658,158.967
C01398=1025.085,183.444,385.158,168.770,47.654,158.967
C01399=1025.091,183.693,385.134,168.772,47.649,158.966
C01400=1025.096,183.942,385.110,168.776,47.645,158.966
C01401=1025.102,184.191,385.088,168.780,47.641,158.966
C01402=1025.107,184.440,385.065,168.784,47.637,158.965
C01403=1025.112,184.689,385.041,168.787,47.633,158.965
C01404=1025.118,184.937,385.017,168.791,47.629,158.964
C01405=1025.123,185.186,384.994,168.795,47.624,158.964
C01406=1025.129,185.435,384.971,168.799,47.620,158.964
C01407=1025.135,185.683,384.947,168.802,47.616,158.963
C01408=1025.140,185.933,384.924,168.805,47.612,158.963
C01409=1025.146,186.182,384.901,168.809,47.608,158.963
C01410=1025.152,186.430,384.877,168.813,47.604,158.962
C01411=1025.157,186.679,384.854,168.816,47.599,158.962
C01412=1025.163,186.928,384.831,168.820,47.595,158.961
C01413=1025.168,187.176,384.806,168.824,47.591,158.961
C01414=1025.174,187.425,384.783,168.828,47.587,158.961
C01415=1025.181,187.708,384.757,168.832,47.582,158.960
C01416=1025.186,187.991,384.730,168.836,47.577,158.960
C01417=1025.193,188.273,384.704,168.840,47.572,158.959
C01418=1025.200,188.556,384.677,168.845,47.568,158.959
C01419=1025.205,188.805,384.653,168.848,47.564,158.959
C01420=1025.211,189.053,384.630,168.852,47.560,158.958
C01421=1025.216,189.302,384.607,168.855,47.556,158.958
C01422=1025.222,189.551,384.583,168.859,47.552,158.958
C01423=1025.227,189.799,384.560,168.863,47.548,158.957
C01424=1025.233,190.048,384.535,168.867,47.543,158.957
C01425=1025.239,190.298,384.512,168.871,47.539,158.957
C01426=1025.245,190.546,384.488,168.874,47.535,158.956
C01427=1025.250,190.795,384.465,168.878,47.531,158.956
C01428=1025.256,191.043,384.441,168.882,47.527,158.956
C01429=1025.262,191.292,384.418,168.886,47.522,158.955
C01430=1025.267,191.541,384.394,168.889,47.518,158.955
C01431=1025.274,191.790,384.371,168.893,47.514,158.955
C01432=1025.279,192.039,384.346,168.897,47.510,158.954
C01433=1025.285,192.288,384.323,168.901,47.506,158.954
C01434=1025.291,192.536,384.300,168.906,47.501,158.953
C01435=1025.296,192.785,384.276,168.909,47.497,158.953
C01436=1025.302,193.034,384.252,168.913,47.493,158.953
C01437=1025.308,193.283,384.228,168.917,47.489,158.952
C01438=1025.313,193.532,384.205,168.921,47.485,158.952
C01439=1025.319,193.780,384.181,168.924,47.480,158.952
C01440=1025.325,194.029,384.157,168.928,47.476,158.951
C01441=1025.331,194.278,384.134,168.932,47.472,158.951
C01442=1025.336,194.527,384.109,168.936,47.468,158.951
C01443=1025.342,194.776,384.087,168.940,47.464,158.950
C01444=1025.349,195.025,384.063,168.944,47.460,158.950
C01445=1025.354,195.273,384.038,168.948,47.456,158.950
C01446=1025.360,195.522,384.015,168.951,47.451,158.949
C01447=1025.366,195.772,383.991,168.955,47.447,158.949
C01448=1025.372,196.020,383.967,168.959,47.443,158.949
C01449=1025.378,196.268,383.943,168.964,47.439,158.948
C01450=1025.383,196.517,383.920,168.968,47.435,158.948
C01451=1025.389,196.766,383.896,168.971,47.431,158.948
C01452=1025.395,197.015,383.872,168.975,47.426,158.947
C01453=1025.401,197.263,383.848,168.979,47.422,158.947
C01454=1025.406,197.513,383.824,168.983,47.418,158.947
C01455=1025.412,197.761,383.800,168.986,47.414,158.946
C01456=1025.419,198.010,383.776,168.990,47.410,158.946
C01457=1025.424,198.259,383.752,168.995,47.406,158.946
C01458=1025.430,198.507,383.728,168.999,47.402,158.945
C01459=1025.436,198.757,383.704,169.003,47.398,158.945
C01460=1025.442,199.005,383.681,169.006,47.393,158.945
C01461=1025.448,199.254,383.657,169.010,47.389,158.944
C01462=1025.454,199.503,383.633,169.014,47.385,158.944
C01463=1025.460,199.751,383.609,169.018,47.381,158.944
C01464=1025.466,200.001,383.584,169.023,47.377,158.943
C01465=1025.471,200.249,383.560,169.027,47.373,158.943
C01466=1025.477,200.497,383.536,169.031,47.369,158.943
C01467=1025.483,200.747,383.512,169.034,47.365,158.942
C01468=1025.488,200.995,383.487,169.038,47.361,158.942
C01469=1025.494,201.245,383.463,169.042,47.357,158.942
C01470=1025.499,201.493,383.439,169.046,47.354,158.942
C01471=1025.505,201.741,383.415,169.050,47.350,158.941
C01472=1025.511,201.991,383.390,169.055,47.346,158.941
C01473=1025.517,202.239,383.366,169.059,47.342,158.941
C01474=1025.523,202.489,383.341,169.063,47.338,158.940
C01475=1025.529,202.736,383.317,169.067,47.334,158.940
C01476=1025.535,202.986,383.292,169.070,47.330,158.940
C01477=1025.540,203.234,383.268,169.074,47.326,158.939
C01478=1025.545,203.483,383.244,169.078,47.322,158.939
C01479=1025.570,204.518,383.142,169.475,47.424,159.012
C01480=1025.580,204.919,383.100,169.481,47.418,159.012
C01481=1025.592,205.320,383.059,169.485,47.413,159.011
C01482=1025.602,205.721,383.017,169.490,47.408,159.011
C01483=1025.613,206.121,382.975,169.495,47.403,159.010
C01484=1025.619,206.370,382.949,169.498,47.400,159.010
C01485=1025.625,206.619,382.923,169.501,47.397,159.010
C01486=1025.632,206.867,382.897,169.504,47.394,159.009
C01487=1025.638,207.115,382.871,169.507,47.391,159.009
C01488=1025.645,207.365,382.845,169.511,47.387,159.009
C01489=1025.652,207.613,382.819,169.514,47.384,159.009
C01490=1025.658,207.861,382.793,169.517,47.381,159.008
C01491=1025.665,208.110,382.767,169.520,47.378,159.008
C01492=1025.671,208.358,382.741,169.523,47.375,159.008
C01493=1025.678,208.607,382.714,169.526,47.372,159.008
C01494=1025.684,208.855,382.688,169.528,47.369,159.007
C01495=1025.691,209.104,382.663,169.531,47.366,159.007
C01496=1025.698,209.353,382.637,169.535,47.363,159.007
C01497=1025.704,209.601,382.610,169.538,47.360,159.007
C01498=1025.711,209.850,382.584,169.541,47.357,159.006
C01499=1025.717,210.098,382.557,169.544,47.354,159.006
C01500=1025.724,210.347,382.532,169.547,47.351,159.006
C01501=1025.731,210.595,382.506,169.550,47.348,159.006
C01502=1025.736,210.844,382.479,169.553,47.345,159.005
C01503=1025.743,211.092,382.453,169.556,47.342,159.005
C01504=1025.749,211.341,382.426,169.560,47.339,159.005
C01505=1025.756,211.590,382.400,169.563,47.336,159.005
C01506=1025.763,211.838,382.374,169.566,47.333,159.005
C01507=1025.769,212.087,382.347,169.569,47.330,159.004
C01508=1025.776,212.335,382.320,169.572,47.327,159.004
C01509=1025.781,212.584,382.295,169.576,47.324,159.004
C01510=1025.788,212.832,382.268,169.579,47.321,159.004
C01511=1025.795,213.080,382.242,169.582,47.318,159.003
C01512=1025.801,213.330,382.215,169.585,47.316,159.003
C01513=1025.808,213.578,382.189,169.588,47.313,159.003
C01514=1025.814,213.827,382.162,169.590,47.310,159.003
C01515=1025.821,214.075,382.136,169.594,47.307,159.002
C01516=1025.828,214.323,382.109,169.597,47.304,159.002
C01517=1025.833,214.572,382.083,169.600,47.301,159.002
C01518=1025.841,214.821,382.056,169.603,47.298,159.002
C01519=1025.846,215.069,382.030,169.606,47.295,159.002
C01520=1025.853,215.318,382.003,169.610,47.292,159.001
C01521=1025.860,215.566,381.977,169.613,47.289,159.001
C01522=1025.866,215.815,381.950,169.616,47.287,159.001
C01523=1025.873,216.062,381.924,169.619,47.284,159.001
C01524=1025.880,216.311,381.897,169.622,47.281,159.001
C01525=1025.887,216.560,381.870,169.625,47.278,159.000
C01526=1025.893,216.808,381.844,169.629,47.275,159.000
C01527=1025.900,217.057,381.817,169.632,47.272,159.000
C01528=1025.906,217.305,381.791,169.635,47.269,159.000
C01529=1025.912,217.554,381.764,169.638,47.266,159.000
C01530=1025.919,217.802,381.738,169.641,47.263,158.999
C01531=1025.926,218.051,381.711,169.645,47.261,158.999
C01532=1025.932,218.299,381.685,169.648,47.258,158.999
C01533=1025.939,218.547,381.658,169.651,47.255,158.999
C01534=1025.946,218.797,381.631,169.655,47.252,158.999
C01535=1025.952,219.045,381.605,169.658,47.249,158.998
C01536=1025.963,219.449,381.561,169.663,47.245,158.998
C01537=1025.973,219.853,381.517,169.668,47.240,158.998
C01538=1025.983,220.257,381.473,169.673,47.235,158.997
C01539=1025.995,220.661,381.430,169.679,47.231,158.997
C01540=1026.000,220.909,381.403,169.681,47.229,158.997
C01541=1026.007,221.158,381.375,169.684,47.226,158.997
C01542=1026.013,221.406,381.349,169.688,47.223,158.997
C01543=1026.020,221.654,381.322,169.691,47.220,158.997
C01544=1026.027,221.903,381.295,169.694,47.217,158.996
C01545=1026.032,222.152,381.268,169.698,47.215,158.996
C01546=1026.040,222.400,381.241,169.701,47.212,158.996
C01547=1026.046,222.649,381.214,169.704,47.210,158.996
C01548=1026.052,222.897,381.187,169.707,47.206,158.996
C01549=1026.059,223.145,381.160,169.711,47.204,158.996
C01550=1026.065,223.394,381.133,169.714,47.201,158.995
C01551=1026.072,223.642,381.106,169.717,47.199,158.995
C01552=1026.078,223.891,381.079,169.720,47.196,158.995
C01553=1026.086,224.139,381.051,169.724,47.193,158.995
C01554=1026.091,224.388,381.025,169.727,47.190,158.995
C01555=1026.098,224.636,380.997,169.730,47.188,158.995
C01556=1026.105,224.885,380.971,169.734,47.185,158.994
C01557=1026.111,225.133,380.943,169.737,47.182,158.994
C01558=1026.118,225.382,380.916,169.740,47.179,158.994
C01559=1026.124,225.630,380.889,169.744,47.177,158.994
C01560=1026.131,225.878,380.862,169.747,47.175,158.994
C01561=1026.138,226.127,380.835,169.750,47.172,158.994
C01562=1026.144,226.376,380.808,169.754,47.169,158.994
C01563=1026.151,226.624,380.781,169.757,47.166,158.993
C01564=1026.157,226.872,380.754,169.760,47.164,158.993
C01565=1026.164,227.121,380.726,169.763,47.161,158.993
C01566=1026.170,227.370,380.699,169.767,47.158,158.993
C01567=1026.177,227.618,380.671,169.770,47.156,158.993
C01568=1026.184,227.866,380.645,169.773,47.153,158.993
C01569=1026.190,228.115,380.618,169.777,47.151,158.992
C01570=1026.197,228.363,380.590,169.780,47.148,158.992
C01571=1026.203,228.611,380.563,169.783,47.145,158.992
C01572=1026.209,228.859,380.535,169.787,47.143,158.992
C01573=1026.216,229.108,380.508,169.790,47.140,158.992
C01574=1026.223,229.357,380.480,169.793,47.138,158.992
C01575=1026.229,229.604,380.453,169.796,47.135,158.992
C01576=1026.235,229.853,380.425,169.799,47.133,158.992
C01577=1026.242,230.102,380.398,169.803,47.130,158.991
C01578=1026.248,230.350,380.370,169.806,47.127,158.991
C01579=1026.255,230.599,380.343,169.809,47.125,158.991
C01580=1026.261,230.847,380.315,169.813,47.123,158.991
C01581=1026.268,231.095,380.287,169.816,47.120,158.991
C01582=1026.274,231.344,380.260,169.820,47.118,158.991
C01583=1026.281,231.593,380.233,169.823,47.115,158.991
C01584=1026.288,231.841,380.205,169.826,47.113,158.991
C01585=1026.294,232.089,380.178,169.830,47.110,158.990
C01586=1026.300,232.337,380.149,169.833,47.108,158.990
C01587=1026.306,232.586,380.122,169.836,47.105,158.990
C01588=1026.313,232.834,380.094,169.840,47.103,158.990
C01589=1026.320,233.083,380.066,169.843,47.101,158.990
C01590=1026.326,233.331,380.038,169.846,47.098,158.990
C01591=1026.332,233.579,380.011,169.850,47.095,158.990
C01592=1026.343,233.976,379.967,169.855,47.092,158.990
C01593=1026.353,234.372,379.922,169.861,47.087,158.989
C01594=1026.364,234.768,379.879,169.866,47.084,158.989
C01595=1026.374,235.164,379.834,169.871,47.080,158.989
C01596=1026.381,235.412,379.806,169.875,47.078,158.989
C01597=1026.387,235.661,379.778,169.878,47.075,158.989
C01598=1026.394,235.909,379.751,169.882,47.073,158.989
C01599=1026.400,236.158,379.722,169.885,47.070,158.989
C01600=1026.407,236.406,379.695,169.888,47.068,158.989
C01601=1026.413,236.655,379.667,169.892,47.065,158.989
C01602=1026.419,236.903,379.640,169.895,47.063,158.989
C01603=1026.426,237.151,379.612,169.898,47.060,158.988
C01604=1026.433,237.399,379.584,169.902,47.058,158.988
C01605=1026.439,237.648,379.556,169.905,47.056,158.988
C01606=1026.445,237.897,379.528,169.909,47.053,158.988
C01607=1026.452,238.144,379.500,169.912,47.051,158.988
C01608=1026.459,238.393,379.472,169.916,47.049,158.988
C01609=1026.466,238.641,379.444,169.919,47.046,158.988
C01610=1026.472,238.890,379.416,169.923,47.044,158.988
C01611=1026.478,239.139,379.388,169.926,47.041,158.988
C01612=1026.485,239.386,379.360,169.929,47.039,158.988
C01613=1026.492,239.635,379.332,169.933,47.037,158.988
C01614=1026.499,239.883,379.304,169.936,47.034,158.988
C01615=1026.505,240.132,379.276,169.940,47.033,158.988
C01616=1026.512,240.380,379.247,169.944,47.030,158.988
C01617=1026.518,240.629,379.219,169.947,47.028,158.987
C01618=1026.524,240.877,379.191,169.950,47.026,158.987
C01619=1026.531,241.125,379.163,169.954,47.023,158.987
C01620=1026.537,241.374,379.135,169.957,47.021,158.987
C01621=1026.544,241.621,379.106,169.961,47.019,158.987
C01622=1026.550,241.870,379.078,169.964,47.017,158.987
C01623=1026.557,242.119,379.050,169.968,47.014,158.987
C01624=1026.563,242.367,379.021,169.971,47.012,158.987
C01625=1026.570,242.615,378.993,169.975,47.010,158.987
C01626=1026.576,242.863,378.964,169.979,47.008,158.987
C01627=1026.583,243.112,378.937,169.982,47.006,158.987
C01628=1026.589,243.360,378.907,169.985,47.003,158.987
C01629=1026.596,243.608,378.880,169.989,47.001,158.987
C01630=1026.603,243.856,378.851,169.992,46.998,158.987
C01631=1026.609,244.105,378.823,169.996,46.997,158.987
C01632=1026.615,244.353,378.794,170.000,46.994,158.987
C01633=1026.622,244.601,378.766,170.003,46.993,158.987
C01634=1026.628,244.850,378.737,170.007,46.990,158.987
C01635=1026.634,245.098,378.708,170.010,46.988,158.987
C01636=1026.640,245.346,378.680,170.014,46.986,158.987
C01637=1026.647,245.594,378.651,170.017,46.984,158.987
C01638=1026.653,245.842,378.622,170.021,46.982,158.987
C01639=1026.659,246.091,378.594,170.025,46.980,158.987
C01640=1026.666,246.339,378.566,170.028,46.977,158.987
C01641=1026.672,246.587,378.536,170.032,46.976,158.987
C01642=1026.678,246.836,378.508,170.035,46.973,158.987
C01643=1026.685,247.084,378.479,170.039,46.971,158.987
C01644=1026.692,247.332,378.451,170.042,46.969,158.987
C01645=1026.698,247.580,378.422,170.046,46.967,158.987
C01646=1026.704,247.829,378.393,170.050,46.965,158.987
C01647=1026.711,248.078,378.364,170.053,46.963,158.987
C01648=1026.721,248.467,378.319,170.058,46.960,158.987
C01649=1026.731,248.857,378.273,170.064,46.956,158.987
C01650=1026.742,249.248,378.229,170.070,46.953,158.987
C01651=1026.751,249.638,378.183,170.076,46.950,158.987
C01652=1026.758,249.886,378.154,170.079,46.948,158.987
C01653=1026.765,250.133,378.126,170.083,46.946,158.987
C01654=1026.771,250.382,378.097,170.086,46.944,158.987
C01655=1026.777,250.630,378.068,170.090,46.942,158.987
C01656=1026.784,250.879,378.039,170.093,46.940,158.987
C01657=1026.791,251.127,378.010,170.097,46.938,158.987
C01658=1026.797,251.375,377.981,170.101,46.936,158.987
C01659=1026.803,251.623,377.952,170.104,46.934,158.987
C01660=1026.809,251.871,377.923,170.108,46.932,158.987
C01661=1026.817,252.120,377.894,170.112,46.930,158.987
C01662=1026.823,252.368,377.865,170.115,46.928,158.987
C01663=1026.829,252.616,377.836,170.119,46.926,158.987
C01664=1026.836,252.864,377.807,170.122,46.924,158.987
C01665=1026.843,253.113,377.779,170.126,46.922,158.987
C01666=1026.850,253.361,377.750,170.130,46.920,158.987
C01667=1026.856,253.609,377.720,170.133,46.918,158.987
C01668=1026.862,253.857,377.691,170.138,46.916,158.987
C01669=1026.870,254.106,377.663,170.141,46.913,158.987
C01670=1026.876,254.354,377.634,170.145,46.912,158.987
C01671=1026.882,254.602,377.605,170.149,46.910,158.987
C01672=1026.889,254.851,377.575,170.152,46.908,158.987
C01673=1026.896,255.099,377.547,170.156,46.906,158.987
C01674=1026.902,255.347,377.518,170.159,46.904,158.987
C01675=1026.908,255.595,377.489,170.163,46.902,158.987
C01676=1026.915,255.844,377.459,170.167,46.900,158.987
C01677=1026.922,256.092,377.430,170.170,46.898,158.987
C01678=1026.929,256.339,377.401,170.174,46.896,158.987
C01679=1026.936,256.588,377.372,170.178,46.894,158.987
C01680=1026.942,256.836,377.343,170.181,46.892,158.987
C01681=1026.949,257.085,377.313,170.185,46.890,158.987
C01682=1026.956,257.333,377.285,170.190,46.888,158.987
C01683=1026.962,257.581,377.256,170.193,46.886,158.987
C01684=1026.969,257.829,377.226,170.197,46.884,158.987
C01685=1026.975,258.077,377.196,170.201,46.883,158.987
C01686=1026.982,258.325,377.168,170.204,46.880,158.987
C01687=1026.989,258.574,377.139,170.208,46.879,158.987
C01688=1026.996,258.822,377.110,170.212,46.877,158.988
C01689=1027.003,259.070,377.079,170.215,46.875,158.988
C01690=1027.009,259.318,377.050,170.219,46.873,158.988
C01691=1027.017,259.567,377.022,170.224,46.871,158.988
C01692=1027.023,259.815,376.993,170.227,46.869,158.988
C01693=1027.029,260.063,376.963,170.231,46.867,158.988
C01694=1027.036,260.311,376.933,170.235,46.865,158.988
C01695=1027.042,260.559,376.904,170.238,46.863,158.988
C01696=1027.050,260.807,376.875,170.242,46.862,158.988
C01697=1027.057,261.056,376.846,170.246,46.860,158.988
C01698=1027.063,261.304,376.815,170.249,46.858,158.988
C01699=1027.069,261.552,376.786,170.253,46.857,158.988
C01700=1027.076,261.800,376.756,170.257,46.855,158.988
C01701=1027.083,262.049,376.727,170.262,46.853,158.988
C01702=1027.089,262.296,376.697,170.265,46.851,158.989
C01703=1027.096,262.545,376.668,170.269,46.849,158.989
C01704=1027.106,262.933,376.621,170.275,46.847,158.989
C01705=1027.116,263.321,376.574,170.280,46.844,158.989
C01706=1027.126,263.710,376.528,170.287,46.841,158.989
C01707=1027.137,264.099,376.481,170.292,46.838,158.989
C01708=1027.143,264.347,376.451,170.296,46.837,158.989
C01709=1027.150,264.595,376.422,170.300,46.835,158.989
C01710=1027.156,264.843,376.392,170.305,46.833,158.989
C01711=1027.164,265.091,376.362,170.308,46.831,158.989
C01712=1027.169,265.340,376.332,170.312,46.830,158.990
C01713=1027.176,265.588,376.302,170.316,46.828,158.990
C01714=1027.183,265.835,376.272,170.320,46.827,158.990
C01715=1027.190,266.083,376.242,170.324,46.825,158.990
C01716=1027.196,266.332,376.213,170.327,46.823,158.990
C01717=1027.203,266.580,376.182,170.331,46.822,158.990
C01718=1027.209,266.828,376.153,170.335,46.820,158.990
C01719=1027.216,267.076,376.122,170.340,46.818,158.990
C01720=1027.223,267.324,376.092,170.343,46.816,158.990
C01721=1027.229,267.573,376.063,170.347,46.815,158.991
C01722=1027.236,267.821,376.033,170.351,46.814,158.991
C01723=1027.242,268.069,376.002,170.355,46.812,158.991
C01724=1027.249,268.317,375.972,170.359,46.810,158.991
C01725=1027.256,268.564,375.942,170.362,46.808,158.991
C01726=1027.262,268.813,375.912,170.366,46.807,158.991
C01727=1027.269,269.061,375.881,170.371,46.805,158.991
C01728=1027.275,269.309,375.851,170.375,46.804,158.991
C01729=1027.282,269.557,375.821,170.379,46.802,158.992
C01730=1027.289,269.805,375.791,170.383,46.801,158.992
C01731=1027.295,270.053,375.761,170.386,46.799,158.992
C01732=1027.302,270.301,375.730,170.390,46.798,158.992
C01733=1027.308,270.549,375.700,170.394,46.796,158.992
C01734=1027.315,270.797,375.670,170.398,46.795,158.992
C01735=1027.322,271.046,375.639,170.403,46.793,158.992
C01736=1027.328,271.293,375.609,170.406,46.791,158.993
C01737=1027.335,271.542,375.579,170.411,46.790,158.993
C01738=1027.341,271.789,375.549,170.414,46.788,158.993
C01739=1027.348,272.038,375.518,170.418,46.787,158.993
C01740=1027.355,272.286,375.487,170.422,46.786,158.993
C01741=1027.361,272.533,375.457,170.426,46.784,158.993
C01742=1027.368,272.782,375.427,170.430,46.783,158.994
C01743=1027.375,273.030,375.396,170.435,46.781,158.994
C01744=1027.381,273.278,375.367,170.439,46.780,158.994
C01745=1027.388,273.526,375.336,170.442,46.778,158.994
C01746=1027.395,273.774,375.305,170.446,46.776,158.994
C01747=1027.401,274.022,375.274,170.450,46.775,158.994
C01748=1027.407,274.270,375.244,170.454,46.774,158.995
C01749=1027.415,274.518,375.213,170.459,46.772,158.995
C01750=1027.421,274.766,375.182,170.463,46.771,158.995
C01751=1027.428,275.014,375.153,170.467,46.770,158.995
C01752=1027.434,275.262,375.122,170.470,46.768,158.995
C01753=1027.441,275.510,375.090,170.475,46.767,158.996
C01754=1027.448,275.758,375.060,170.478,46.765,158.996
C01755=1027.454,276.006,375.030,170.483,46.764,158.996
C01756=1027.461,276.254,374.999,170.487,46.762,158.996
C01757=1027.468,276.502,374.968,170.491,46.761,158.996
C01758=1027.474,276.750,374.937,170.495,46.759,158.996
C01759=1027.482,276.998,374.907,170.499,46.758,158.997
C01760=1027.492,277.392,374.858,170.506,46.756,158.997
C01761=1027.503,277.785,374.809,170.513,46.754,158.997
C01762=1027.513,278.178,374.760,170.518,46.752,158.998
C01763=1027.523,278.571,374.711,170.526,46.750,158.998
C01764=1027.530,278.819,374.680,170.529,46.748,158.998
C01765=1027.537,279.067,374.649,170.533,46.747,158.998
C01766=1027.543,279.315,374.618,170.537,46.746,158.999
C01767=1027.549,279.562,374.587,170.541,46.745,158.999
C01768=1027.556,279.811,374.556,170.546,46.743,158.999
C01769=1027.563,280.059,374.524,170.550,46.742,158.999
C01770=1027.569,280.307,374.493,170.554,46.741,158.999
C01771=1027.576,280.555,374.463,170.558,46.740,159.000
C01772=1027.583,280.803,374.431,170.562,46.738,159.000
C01773=1027.589,281.050,374.400,170.567,46.737,159.000
C01774=1027.596,281.299,374.370,170.571,46.736,159.000
C01775=1027.602,281.547,374.338,170.575,46.735,159.001
C01776=1027.609,281.794,374.307,170.579,46.734,159.001
C01777=1027.616,282.042,374.275,170.583,46.732,159.001
C01778=1027.622,282.291,374.245,170.588,46.731,159.001
C01779=1027.630,282.538,374.214,170.592,46.730,159.002
C01780=1027.636,282.786,374.182,170.596,46.729,159.002
C01781=1027.643,283.034,374.151,170.600,46.727,159.002
C01782=1027.650,283.282,374.120,170.604,46.726,159.002
C01783=1027.657,283.530,374.088,170.609,46.724,159.002
C01784=1027.663,283.779,374.057,170.613,46.723,159.003
C01785=1027.670,284.026,374.026,170.617,46.722,159.003
C01786=1027.676,284.274,373.995,170.621,46.721,159.003
C01787=1027.684,284.522,373.964,170.626,46.720,159.004
C01788=1027.691,284.770,373.932,170.630,46.719,159.004
C01789=1027.697,285.018,373.901,170.634,46.718,159.004
C01790=1027.704,285.266,373.869,170.638,46.717,159.004
C01791=1027.711,285.514,373.838,170.643,46.715,159.005
C01792=1027.718,285.761,373.807,170.647,46.714,159.005
C01793=1027.724,286.009,373.775,170.651,46.713,159.005
C01794=1027.731,286.257,373.744,170.655,46.712,159.005
C01795=1027.738,286.505,373.712,170.660,46.711,159.006
C01796=1027.744,286.753,373.681,170.664,46.710,159.006
C01797=1027.751,287.001,373.649,170.668,46.709,159.006
C01798=1027.758,287.249,373.618,170.673,46.708,159.006
C01799=1027.764,287.497,373.586,170.678,46.706,159.007
C01800=1027.771,287.744,373.554,170.682,46.705,159.007
C01801=1027.778,287.992,373.522,170.686,46.704,159.007
C01802=1027.784,288.240,373.491,170.690,46.703,159.008
C01803=1027.791,288.488,373.459,170.695,46.702,159.008
C01804=1027.798,288.736,373.428,170.699,46.701,159.008
C01805=1027.805,288.983,373.396,170.703,46.700,159.008
C01806=1027.811,289.232,373.364,170.708,46.699,159.009
C01807=1027.818,289.479,373.332,170.712,46.698,159.009
C01808=1027.824,289.727,373.301,170.716,46.697,159.009
C01809=1027.832,289.975,373.268,170.720,46.696,159.010
C01810=1027.839,290.223,373.237,170.725,46.695,159.010
C01811=1027.845,290.471,373.205,170.730,46.694,159.010
